// SIMATIC S7-200 project (STEP 7-Micro/WIN), CPU 224XP IE REL 02.01

SYMBOL_TABLE DI采集
急停               V0.0
单机/联机            V0.1
油泵启停             V0.2
1#进油启/停          V0.3
1#回油启/停          V0.4
2#进油启/停          V0.5
2#回油启/停          V0.6
缺相保护             V0.7
输入备用             V1.0
END_SYMBOL_TABLE

SYMBOL_TABLE DO控制
油泵_启             V22.0
1#进油_启           V20.2
1#回油_启           V20.4
1#卸荷_启           V20.6
2#进油_启           V21.0
2#回油_启           V21.2
2#卸荷_启           V21.4
备用_启             V21.6
油泵_停             V22.1
1#进油_停           V20.3
1#回油_停           V20.5
1#卸荷_停           V20.7
2#进油_停           V21.1
2#回油_停           V21.3
2#卸荷_停           V21.5
备用_停             V21.7
油泵_同             V41.0
1#进油_同           V40.1
1#回油_同           V40.2
1#卸荷_同           V40.3
2#进油_同           V40.4
2#回油_同           V40.5
2#卸荷_同           V40.6
备用_同             V40.7
END_SYMBOL_TABLE

SYMBOL_TABLE AI采集
AI1备用            VW50
AI2备用            VW52
1#压力             VW54
1#位移             VW56
2#压力             VW58
2#位移             VW60
压力1KN            VD78
压力2KN            VD86
压力量程上限           VW2000
位移量程上限           VW2002
AI1上限            VW2050
AI1下限            VW2052
AI2上限            VW2054
AI2下限            VW2056
1#压力L上限          VW2058
1#压力L下限          VW2060
1#位移L上限          VW2062
1#位移L下限          VW2064
2#压力L上限          VW2066
2#压力L下限          VW2068
2#位移L上限          VW2070
2#位移L下限          VW2072
AI1备用C           VW150
AI2备用C           VW152
1#压力C            VW154
1#位移C            VW156
2#压力C            VW158
2#位移C            VW160
1#压力断线           V100.0
1#位移断线           V100.1
2#压力断线           V100.2
2#位移断线           V100.3
END_SYMBOL_TABLE

SYMBOL_TABLE 故障
本机安全极限压力         VW2004
本机安全极限位移         VW2006
补压压力             VW2008
同步位移             VW2010
回程允许时间           VW2012
回程停机位移           VW2014
1#超本机压力_A        V2210.0
1#超本机位移_A        V2210.1
2#超本机压力_A        V2210.2
2#超本机位移_A        V2210.3
1#超安全压力_A        V2210.4
2#超安全压力_A        V2210.5
1#回程故障_A         V2210.6
2#回程故障_A         V2210.7
1#压力断线_A         V2211.0
1#位移断线_A         V2211.1
2#压力断线_A         V2211.2
2#位移断线_A         V2211.3
电机故障_A           V2211.4
总故障_A            V2211.7
END_SYMBOL_TABLE

SYMBOL_TABLE A1
A1设备标志           VW4018
A1第1B            VW4020
A1第2B            VW4022
A1第3B            VW4024
A1第4B            VW4026
A1第5B            VW4028
A1第6B            VW4030
A1终张B            VW4032
A1超张B            VW4034
A1回程B            VW4036
A1第1Y            VW4038
A1第2Y            VW4040
A1第3_1Y          VW4042
A1第3_2Y          VW4044
A1第4_1Y          VW4046
A1第4_2Y          VW4048
A1第5_1Y          VW4050
A1第5_2Y          VW4052
A1第6_1Y          VW4054
A1第6_2Y          VW4056
A1终张Y            VW4058
A1超张Y            VW4060
A1回程Y            VW4062
A1第1W            VW4064
A1第2W            VW4066
A1第3_1W          VW4068
A1第3_2W          VW4070
A1第4_1W          VW4072
A1第4_2W          VW4074
A1第5_1W          VW4076
A1第5_2W          VW4078
A1第6_1W          VW4080
A1第6_2W          VW4082
A1终张W            VW4084
A1超张W            VW4086
A1回程W            VW4088
A1安全B            VW4090
A1安全TJM          VW4092
A1设计油压M          VW4094
A1单根张拉力          VW4098
A1孔根数            VW4100
A1理论总伸长量         VW4102
A1理论总伸长上限        VW4104
A1理论总伸长下限        VW4106
A1实际伸长_mm        VW4112
A1单实际伸长_mm       VW4114
A1自控回程位移         VW4116
A1超张模式           VW4118
A1几次终张           VW4120
A1几顶拉            VW4122
A1顶选择            VW4124
A1是否终张           VW4126
A1理论回缩量（mm）      VW4128
A1张拉位置           VW4136
A1张拉控制力          VD4154
A1Y第1B           VW1300
A1Y第2B           VW1302
A1Y第3B           VW1304
A1Y第4B           VW1306
A1Y第5B           VW1308
A1Y第6B           VW1310
A1Y终张B           VW1312
A1Y超张B           VW1314
A1Y回程B           VW1316
A1Y安全B           VW1318
A1触发记录压力         VW2350
END_SYMBOL_TABLE

SYMBOL_TABLE 主控
卸荷完触发回程          M3.0
有卸荷标志            M1.0
回程停机缓冲位移         VW2016
伸长量不符合           V2212.3
参与机子到目标          V2220.0
A1_设置选择          V3124.0
B1_设置选择          V3124.1
A2_设置选择          V3124.2
B2_设置选择          V3124.3
持荷倒计时            VW2300
张拉位置最小值          VW2302
1组对拉位移最小值        VW2304
2组对拉位移最小值        VW2306
A1目标压力           VW2308
B1目标压力           VW2310
A2目标压力           VW2312
B2目标压力           VW2314
张拉中              V2206.0
回程中              V2206.1
持荷中              V2206.2
卸荷中              V2206.3
有无卸荷             VW2038
倒顶目标标志           V2212.0  // 1为第一次，0为第二进入
持荷完成标志           V2212.1
触发回程             V2212.2
A1伸长量不符合         V2212.4
B1伸长量不符合         V2212.5
A2伸长量不符合         V2212.6
B2伸长量不符合         V2212.7
位移超长触发回程         V2213.0
伸长量高于上限          V2213.1
A1伸长量高于上限        V2213.2
B1伸长量高于上限        V2213.3
A2伸长量高于上限        V2213.4
B2伸长量高于上限        V2213.5
算伸长量             V2213.6
伸长量已反算           V2213.7
自动进油_启           V2214.0
自动回油_启           V2214.1
自动卸荷_启           V2214.2
自动进油_停           V2215.0
自动回油_停           V2215.1
自动卸荷_停           V2215.2
自动进油_出           V2216.0
自动回油_出           V2216.1
自动卸荷_出           V2216.2
A1_实际选择          V2200.0
B1_实际选择          V2200.1
A2_实际选择          V2200.2
B2_实际选择          V2200.3
自动张拉             V2202.0
暂停张拉             V2202.1
手动进油             V2202.2
手动回油             V2202.3
A1到目标标志          V2218.0
B1到目标标志          V2218.1
A2到目标标志          V2218.2
B2到目标标志          V2218.3
A1自动进油_启         V2222.0
A1自动回油_启         V2222.1
A2自动进油_启         V2222.2
A2自动回油_启         V2222.3
A1自动进油_停         V2224.0
A1自动回油_停         V2224.1
A2自动进油_停         V2224.2
A2自动回油_停         V2224.3
A1自动卸荷_启         V2222.4
A2自动卸荷_启         V2222.5
A1自动卸荷_停         V2224.4
A2自动卸荷_停         V2224.5
A1自动进油_输出        V2226.0
A1自动回油_输出        V2226.1
A2自动进油_输出        V2226.2
A2自动回油_输出        V2226.3
A1自动卸荷_输出        V2226.4
A2自动卸荷_输出        V2226.5
A1回程到位           V2230.0
B1回程到位           V2230.1
A2回程到位           V2230.2
B2回程到位           V2230.3
A1卸荷到位           V2420.0
B1卸荷到位           V2420.1
A2卸荷到位           V2420.2
B2卸荷到位           V2420.3
总卸荷到位            V2420.4
A1触发记录           V2232.0
B1触发记录           V2232.1
A2触发记录           V2232.2
B2触发记录           V2232.3
触发写配方            V2232.4  // 触摸屏写完复位
调入已张拉的数据         V2204.0
新数据              V2204.1
调入模板数据           V2204.2
调入已张拉的数据_清       V2204.3
新数据_清            V2204.4
调入模板数据_清         V2204.5
调入已张拉的数据_触发      V2204.6
新数据_触发           V2204.7
调入模板数据_触发        V2205.0
总调入数据            V2205.7
A1回程触发           V2252.0
B1回程触发           V2252.1
A2回程触发           V2252.2
B2回程触发           V2252.3
复位超伸长量上限         V2250.0
复位超伸长量下限         V2250.1
持荷完成标志自锁2S       V2250.2
第一组实伸长量          VW2360
第二组实伸长量          VW2362
下载数据计时           VW2328
持荷时间             T37
张拉过标志            T38
回油时间             T39
故障复位时间           T40
写数据时间            T41
下载数据计时T          T42
持荷完成标志自锁2ST      T43
B1力值             VD2370
B2力值             VD2374
张回程完成标志          V2240.0
主启动油泵            V2254.0
主停止油泵            V2254.1
凋数据序号1           VW2390
凋数据序号2           VW2392
凋数据序号3           VW2394
凋数据序号4           VW2396
凋数据序号            VW2398
调入次数             VW2400
保存数据             V2208.0
不保存数据回程          V2208.1
未完成张拉保存数据回程      V2208.2
完成张拉超张保存数据回      V2208.3
触摸屏修改钢绞线根数       V2404.0
触摸屏修改张拉最大位移      V2404.1
触摸屏修改AB1伸长量      V2404.2
触摸屏修改AB2伸长量      V2404.3
单机频率             VW2120
张拉频率             VW2122
接近目标%            VW2124
目标频率%            VW2126
输出频率             VW2128
接近目标力            VD2130
副机张拉频率           VW2134
A1位移修正           VW2022
B1位移修正           VW2024
A2位移修正           VW2026
B2位移修正           VW2028
A1位移修正触发         VW2030
B1位移修正触发         VW2032
A2位移修正触发         VW2034
B2位移修正触发         VW2036
END_SYMBOL_TABLE

SYMBOL_TABLE 公共存储
G设备标志            VW3018
G第1B             VW3020
G第2B             VW3022
G第3B             VW3024
G第4B             VW3026
G第5B             VW3028
G第6B             VW3030
G终张B             VW3032
G超张B             VW3034
G回程B             VW3036
G第1Y             VW3038
G第2Y             VW3040
G第3_1Y           VW3042
G第3_2Y           VW3044
G第4_1Y           VW3046
G第4_2Y           VW3048
G第5_1Y           VW3050
G第5_2Y           VW3052
G第6_1Y           VW3054
G第6_2Y           VW3056
G终张Y             VW3058
G超张Y             VW3060
G回程Y             VW3062
G第1W             VW3064
G第2W             VW3066
G第3_1W           VW3068
G第3_2W           VW3070
G第4_1W           VW3072
G第4_2W           VW3074
G第5_1W           VW3076
G第5_2W           VW3078
G第6_1W           VW3080
G第6_2W           VW3082
G终张W             VW3084
G超张W             VW3086
G回程W             VW3088
G安全B             VW3090
G安全TJM           VW3092
G设计油压M           VW3094
G                VW3096
G单根张拉力           VW3098
G孔根数             VW3100
G理论总伸长量          VW3102
G理论总伸长上限         VW3104
G理论总伸长下限         VW3106
G实际伸长_mm         VW3112
G单实际伸长_mm        VW3114
G自控回程位移          VW3116
G超张模式            VW3118
G几次终张            VW3120
G几顶拉             VW3122   // 单拉 1对拉 2对拉
G顶选择             VW3124
G是否终张            VW3126
G理论回缩量（mm）       VW3128
G张拉控制力           VD3154
END_SYMBOL_TABLE

SYMBOL_TABLE B1
B1设备标志           VW4418
B1第1B            VW4420
B1第2B            VW4422
B1第3B            VW4424
B1第4B            VW4426
B1第5B            VW4428
B1第6B            VW4430
B1终张B            VW4432
B1超张B            VW4434
B1回程B            VW4436
B1第1Y            VW4438
B1第2Y            VW4440
B1第3_1Y          VW4442
B1第3_2Y          VW4444
B1第4_1Y          VW4446
B1第4_2Y          VW4448
B1第5_1Y          VW4450
B1第5_2Y          VW4452
B1第6_1Y          VW4454
B1第6_2Y          VW4456
B1终张Y            VW4458
B1超张Y            VW4460
B1回程Y            VW4462
B1第1W            VW4464
B1第2W            VW4466
B1第3_1W          VW4468
B1第3_2W          VW4470
B1第4_1W          VW4472
B1第4_2W          VW4474
B1第5_1W          VW4476
B1第5_2W          VW4478
B1第6_1W          VW4480
B1第6_2W          VW4482
B1终张W            VW4484
B1超张W            VW4486
B1回程W            VW4488
B1安全B            VW4490
B1安全TJM          VW4492
B1设计油压M          VW4494
B1单根张拉力          VW4498
B1孔根数            VW4500
B1理论总伸长量         VW4502
B1理论总伸长上限        VW4504
B1理论总伸长下限        VW4506
B1实际伸长_mm        VW4512
B1单实际伸长_mm       VW4514
B1自控回程位移         VW4516
B1超张模式           VW4518
B1几次终张           VW4520
B1几顶拉            VW4522
B1顶选择            VW4524
B1是否终张           VW4526
B1理论回缩量（mm）      VW4528
B1张拉控制力          VD4554
B1#压力            VW2610
B1#位移            VW2612
B2#压力            VW2614
B2#位移            VW2616
B1触发记录压力         VW2352
END_SYMBOL_TABLE

SYMBOL_TABLE A2
A2设备标志           VW4818
A2第1B            VW4820
A2第2B            VW4822
A2第3B            VW4824
A2第4B            VW4826
A2第5B            VW4828
A2第6B            VW4830
A2终张B            VW4832
A2超张B            VW4834
A2回程B            VW4836
A2第1Y            VW4838
A2第2Y            VW4840
A2第3_1Y          VW4842
A2第3_2Y          VW4844
A2第4_1Y          VW4846
A2第4_2Y          VW4848
A2第5_1Y          VW4850
A2第5_2Y          VW4852
A2第6_1Y          VW4854
A2第6_2Y          VW4856
A2终张Y            VW4858
A2超张Y            VW4860
A2回程Y            VW4862
A2第1W            VW4864
A2第2W            VW4866
A2第3_1W          VW4868
A2第3_2W          VW4870
A2第4_1W          VW4872
A2第4_2W          VW4874
A2第5_1W          VW4876
A2第5_2W          VW4878
A2第6_1W          VW4880
A2第6_2W          VW4882
A2终张W            VW4884
A2超张W            VW4886
A2回程W            VW4888
A2安全B            VW4890
A2安全TJM          VW4892
A2设计油压M          VW4894
A2单根张拉力          VW4898
A2孔根数            VW4900
A2理论总伸长量         VW4902
A2理论总伸长上限        VW4904
A2理论总伸长下限        VW4906
A2实际伸长_mm        VW4912
A2单实际伸长_mm       VW4914
A2自控回程位移         VW4916
A2超张模式           VW4918
A2几次终张           VW4920
A2几顶拉            VW4922
A2顶选择            VW4924
A2是否终张           VW4926
A2理论回缩量（mm）      VW4928
A2张拉位置           VW4936
A2张拉控制力          VD4954
A2触发记录压力         VW2354
END_SYMBOL_TABLE

SYMBOL_TABLE B2
B2设备标志           VW5218
B2第1B            VW5220
B2第2B            VW5222
B2第3B            VW5224
B2第4B            VW5226
B2第5B            VW5228
B2第6B            VW5230
B2终张B            VW5232
B2超张B            VW5234
B2回程B            VW5236
B2第1Y            VW5238
B2第2Y            VW5240
B2第3_1Y          VW5242
B2第3_2Y          VW5244
B2第4_1Y          VW5246
B2第4_2Y          VW5248
B2第5_1Y          VW5250
B2第5_2Y          VW5252
B2第6_1Y          VW5254
B2第6_2Y          VW5256
B2终张Y            VW5258
B2超张Y            VW5260
B2回程Y            VW5262
B2第1W            VW5264
B2第2W            VW5266
B2第3_1W          VW5268
B2第3_2W          VW5270
B2第4_1W          VW5272
B2第4_2W          VW5274
B2第5_1W          VW5276
B2第5_2W          VW5278
B2第6_1W          VW5280
B2第6_2W          VW5282
B2终张W            VW5284
B2超张W            VW5286
B2回程W            VW5288
B2安全B            VW5290
B2安全TJM          VW5292
B2设计油压M          VW5294
B2单根张拉力          VW5298
B2孔根数            VW5300
B2理论总伸长量         VW5302
B2理论总伸长上限        VW5304
B2理论总伸长下限        VW5306
B2实际伸长_mm        VW5312
B2单实际伸长_mm       VW5314
B2自控回程位移         VW5316
B2超张模式           VW5318
B2几次终张           VW5320
B2几顶拉            VW5322
B2顶选择            VW5324
B2是否终张           VW5326
B2理论回缩量（mm）      VW5328
B2张拉位置           VW5336
B2张拉控制力          VD5354
B2触发记录压力         VW2356
END_SYMBOL_TABLE

SYMBOL_TABLE mm
密码总错误            V8092.7
当前大于有效           V8092.2
当前小于记忆           V8092.1
有效年              VW8050
有效月              VW8052
有效日              VW8054
记忆年              VW8056
记忆月              VW8058
记忆日              VW8060
当前年              VW8062
当前月              VW8064
当前日              VW8066
校验错误             V8092.0
END_SYMBOL_TABLE

SYMBOL_TABLE 主副交换
副机通讯故障           V2402.1
B1到目标            V2604.0
B2到目标            V2604.1
FB1回程到位          V2604.2
FB2回程到位          V2604.3
B1卸荷到位F          V2604.4
B2卸荷到位F          V2604.5
B1目标%            VW2322
B2目标%            VW2326
触发回程位移           VW2018
B1安全压力           VW1418
B2安全压力           VW1618
F急停              V2600.0
单机_联机F           V2600.1
副油泵启动            V2600.2
副1进油启_停          V2600.3
F1回油启_停          V2600.4
F2进油启_停          V2600.5
F2回油启_停          V2600.6
F缺相保护            V2600.7
F油泵_Y            V2601.0
F1进油_Y           V2601.1
F1回油_Y           V2601.2
F1卸荷_Y           V2601.3
F2进油_Y           V2601.4
F2回油_Y           V2601.5
F2卸荷_Y           V2601.6
F备用_Y            V2601.7
END_SYMBOL_TABLE

SYMBOL_TABLE S7-200 符号
Always_On        SM0.0    // 始终接通为 ON
First_Scan_On    SM0.1    // 仅第一个扫描周期中接通为 ON
Clock_1s         SM0.5    // 在 1 秒钟的循环周期内，接通为 ON 0.5 秒，关断为 OFF 0.5  秒
Time_0_Intrvl    SMB34    // 定时中断 0 的时间间隔（从 1 至 255，以 1 毫秒为增量）。
END_SYMBOL_TABLE

ORGANIZATION_BLOCK 程序块:OB1
TITLE=程序注释
BEGIN
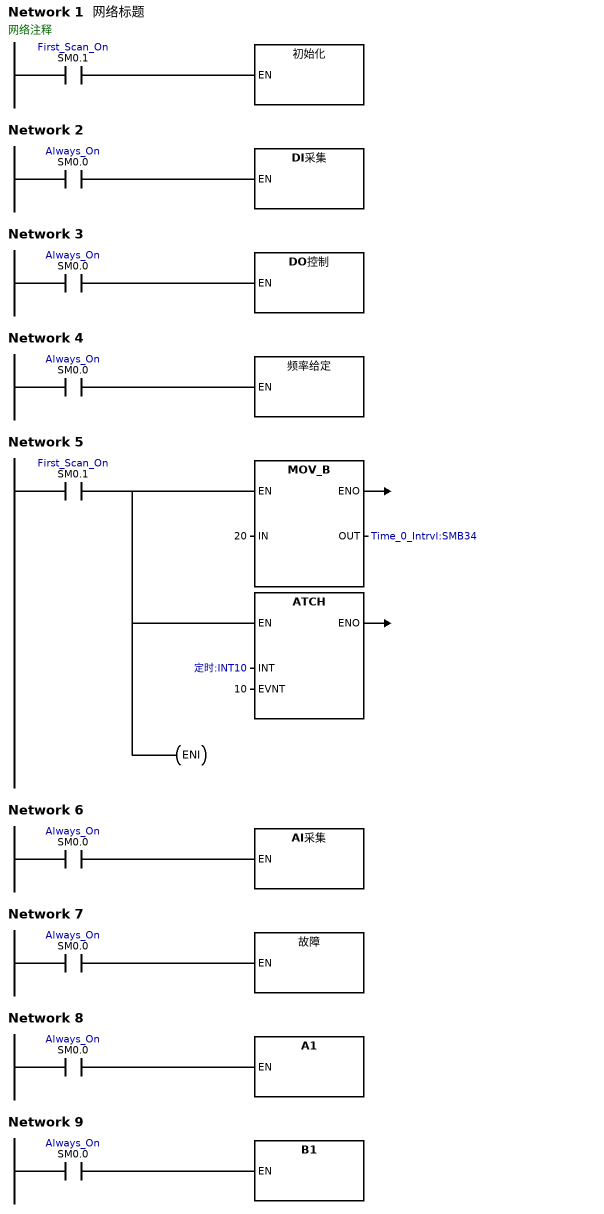
Network 1 // 网络标题
// 网络注释
LD     First_Scan_On:SM0.1
CALL   初始化:SBR0
Network 2
LD     Always_On:SM0.0
CALL   DI采集:SBR1
Network 3
LD     Always_On:SM0.0
CALL   DO控制:SBR2
Network 4
LD     Always_On:SM0.0
CALL   频率给定:SBR30
Network 5
LD     First_Scan_On:SM0.1
MOVB   20, Time_0_Intrvl:SMB34
ATCH   定时:INT10, 10
ENI
Network 6
LD     Always_On:SM0.0
CALL   AI采集:SBR3
Network 7
LD     Always_On:SM0.0
CALL   故障:SBR6
Network 8
LD     Always_On:SM0.0
CALL   A1:SBR7
Network 9
LD     Always_On:SM0.0
CALL   B1:SBR8
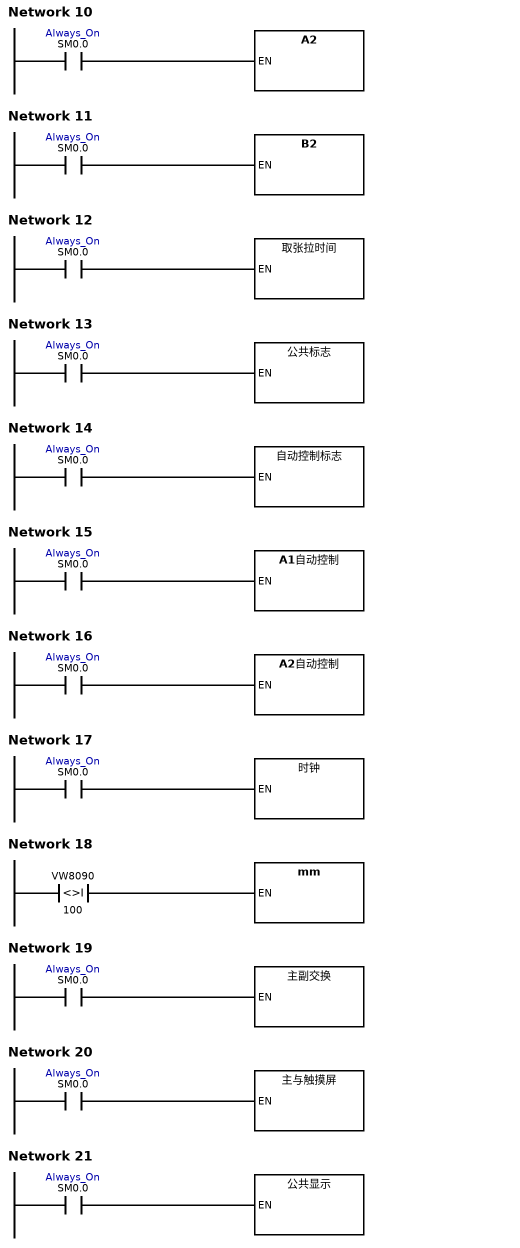
Network 10
LD     Always_On:SM0.0
CALL   A2:SBR9
Network 11
LD     Always_On:SM0.0
CALL   B2:SBR10
Network 12
LD     Always_On:SM0.0
CALL   取张拉时间:SBR28
Network 13
LD     Always_On:SM0.0
CALL   公共标志:SBR13
Network 14
LD     Always_On:SM0.0
CALL   自动控制标志:SBR14
Network 15
LD     Always_On:SM0.0
CALL   A1自动控制:SBR19
Network 16
LD     Always_On:SM0.0
CALL   A2自动控制:SBR20
Network 17
LD     Always_On:SM0.0
CALL   时钟:SBR21
Network 18
LDW<>  VW8090, 100
CALL   mm:SBR22
Network 19
LD     Always_On:SM0.0
CALL   主副交换:SBR23
Network 20
LD     Always_On:SM0.0
CALL   主与触摸屏:SBR18
Network 21
LD     Always_On:SM0.0
CALL   公共显示:SBR24
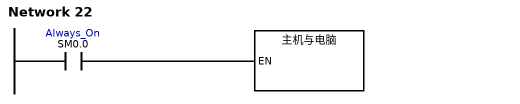
Network 22
LD     Always_On:SM0.0
CALL   主机与电脑:SBR29
END_ORGANIZATION_BLOCK

SUBROUTINE_BLOCK 初始化:SBR0
TITLE=
BEGIN
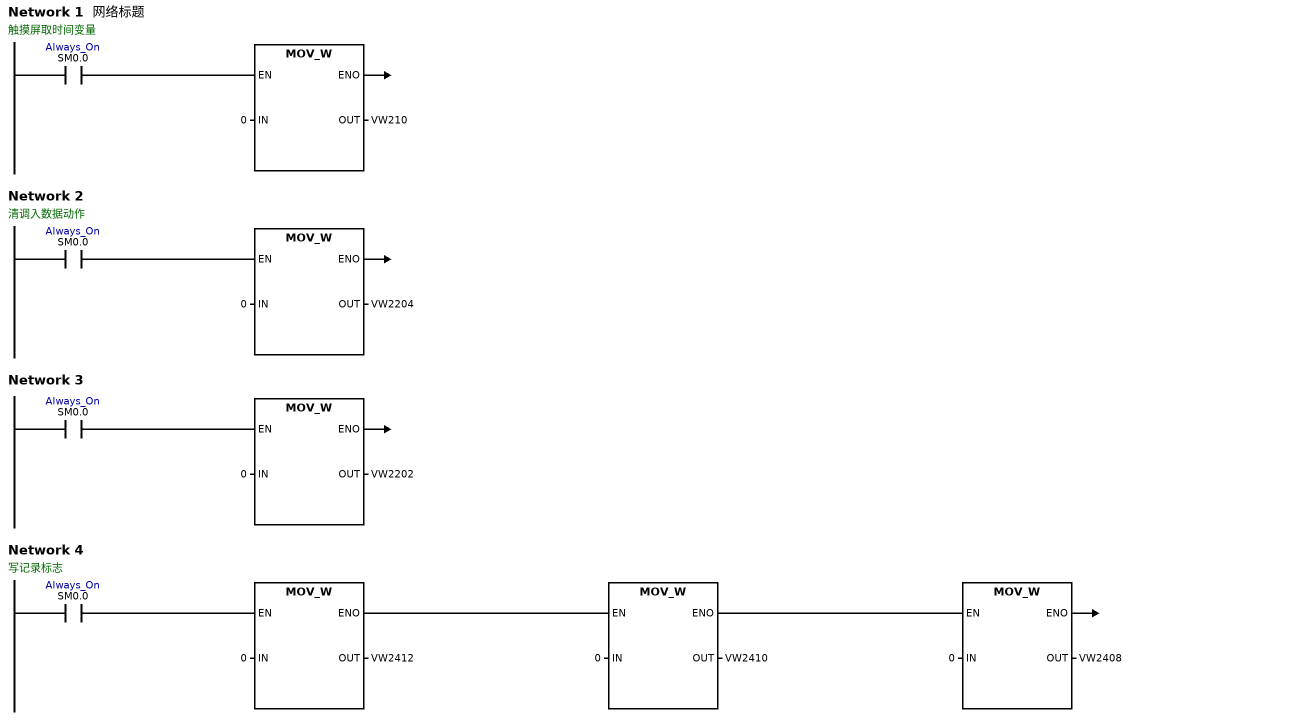
Network 1 // 网络标题
// 触摸屏取时间变量
LD     Always_On:SM0.0
MOVW   0, VW210
Network 2
// 清调入数据动作
LD     Always_On:SM0.0
MOVW   0, VW2204
Network 3
LD     Always_On:SM0.0
MOVW   0, VW2202
Network 4
// 写记录标志
LD     Always_On:SM0.0
MOVW   0, VW2412
AENO
MOVW   0, VW2410
AENO
MOVW   0, VW2408
END_SUBROUTINE_BLOCK

SUBROUTINE_BLOCK DI采集:SBR1
TITLE=
BEGIN
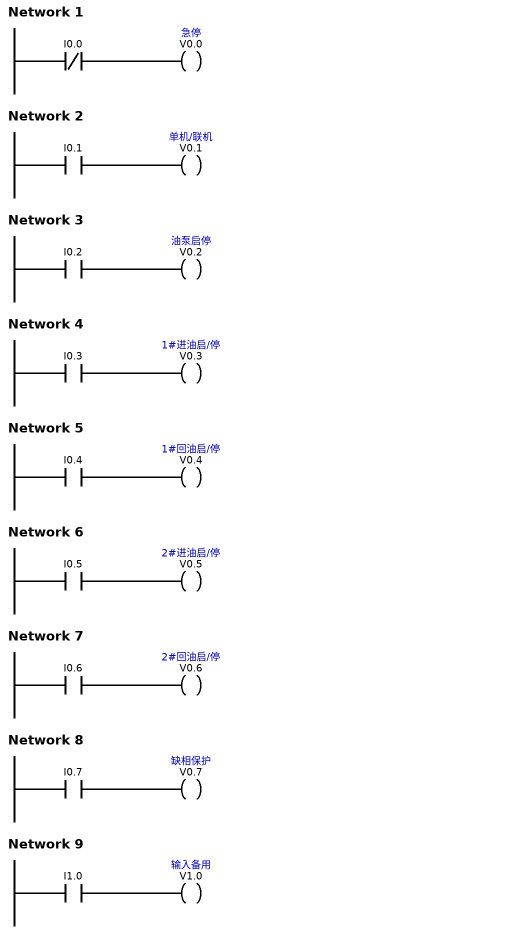
Network 1
LDN    I0.0
=      急停:V0.0
Network 2
LD     I0.1
=      单机/联机:V0.1
Network 3
LD     I0.2
=      油泵启停:V0.2
Network 4
LD     I0.3
=      1#进油启/停:V0.3
Network 5
LD     I0.4
=      1#回油启/停:V0.4
Network 6
LD     I0.5
=      2#进油启/停:V0.5
Network 7
LD     I0.6
=      2#回油启/停:V0.6
Network 8
LD     I0.7
=      缺相保护:V0.7
Network 9
LD     I1.0
=      输入备用:V1.0
END_SUBROUTINE_BLOCK

SUBROUTINE_BLOCK DO控制:SBR2
TITLE=
BEGIN
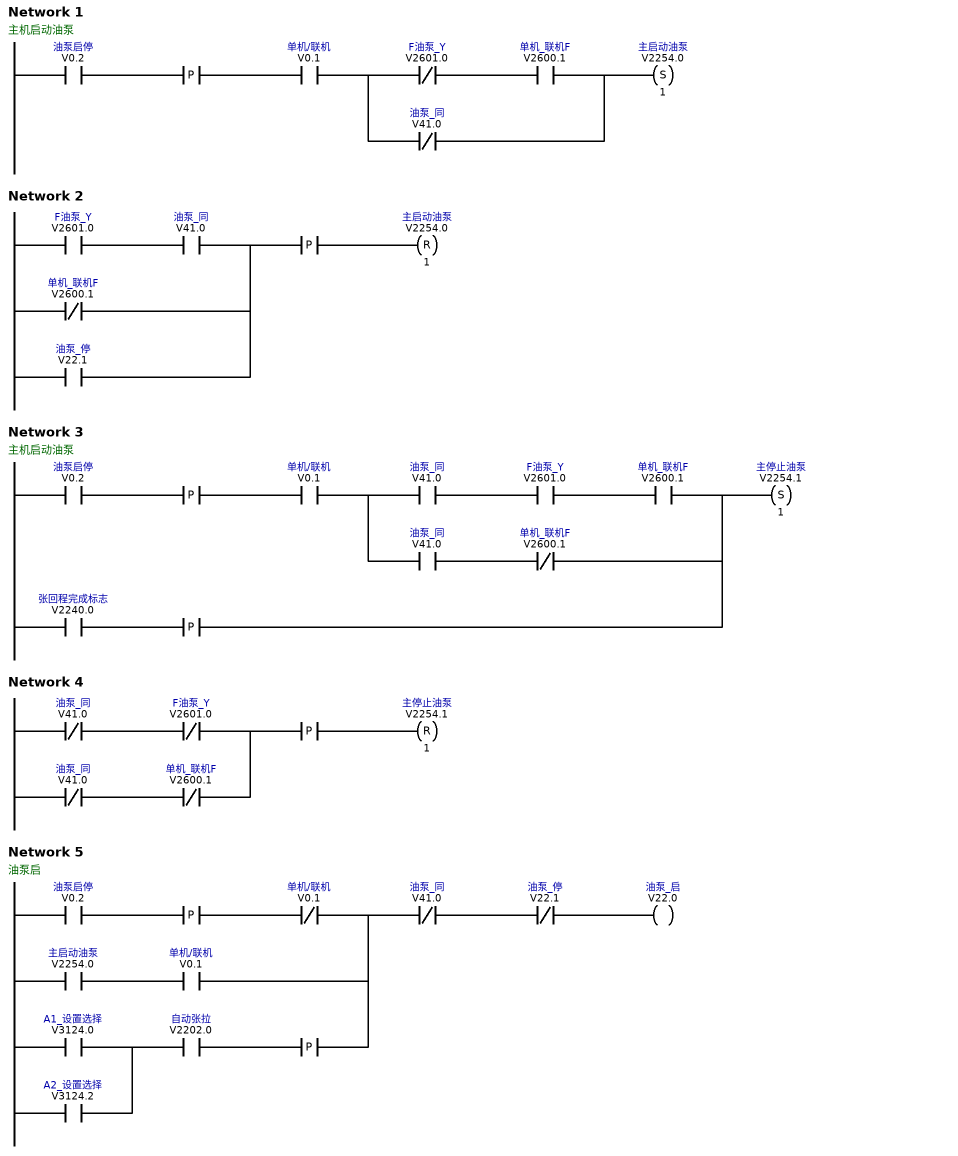
Network 1
// 主机启动油泵
LD     油泵启停:V0.2
EU
A      单机/联机:V0.1
LDN    F油泵_Y:V2601.0
A      单机_联机F:V2600.1
ON     油泵_同:V41.0
ALD
S      主启动油泵:V2254.0, 1
Network 2
LD     F油泵_Y:V2601.0
A      油泵_同:V41.0
ON     单机_联机F:V2600.1
O      油泵_停:V22.1
EU
R      主启动油泵:V2254.0, 1
Network 3
// 主机启动油泵
LD     油泵启停:V0.2
EU
A      单机/联机:V0.1
LD     油泵_同:V41.0
A      F油泵_Y:V2601.0
A      单机_联机F:V2600.1
LD     油泵_同:V41.0
AN     单机_联机F:V2600.1
OLD
ALD
LD     张回程完成标志:V2240.0
EU
OLD
S      主停止油泵:V2254.1, 1
Network 4
LDN    油泵_同:V41.0
AN     F油泵_Y:V2601.0
LDN    油泵_同:V41.0
AN     单机_联机F:V2600.1
OLD
EU
R      主停止油泵:V2254.1, 1
Network 5
// 油泵启
LD     油泵启停:V0.2
EU
AN     单机/联机:V0.1
LD     主启动油泵:V2254.0
A      单机/联机:V0.1
OLD
LD     A1_设置选择:V3124.0
O      A2_设置选择:V3124.2
A      自动张拉:V2202.0
EU
OLD
AN     油泵_同:V41.0
AN     油泵_停:V22.1
=      油泵_启:V22.0
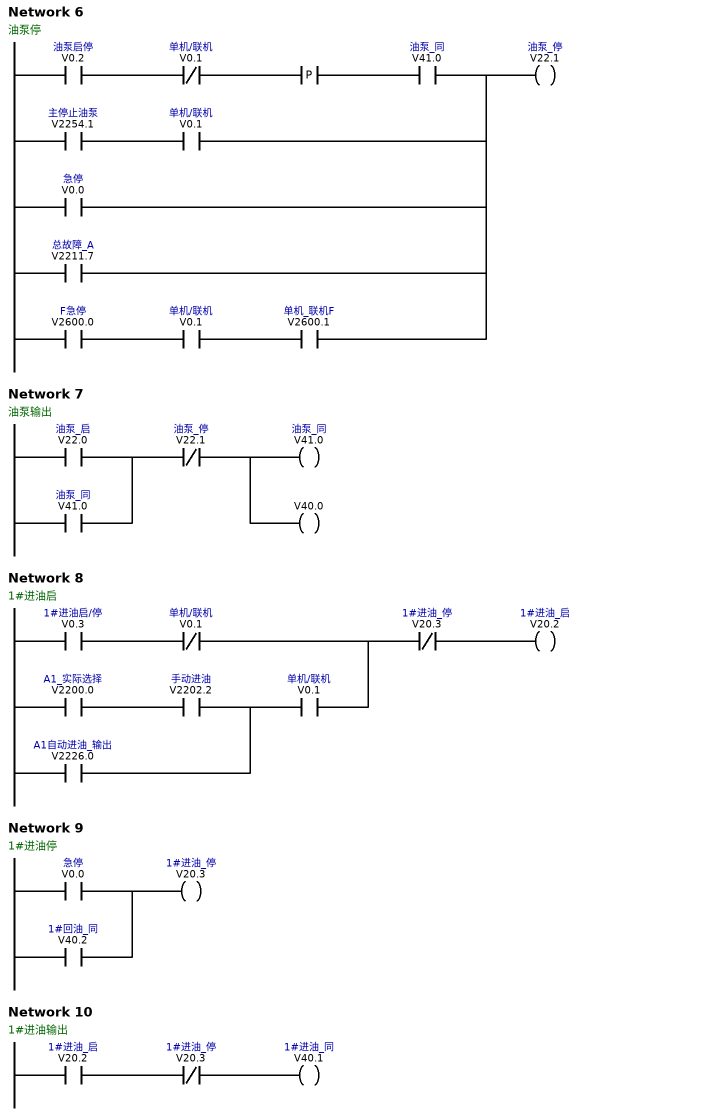
Network 6
// 油泵停
LD     油泵启停:V0.2
AN     单机/联机:V0.1
EU
A      油泵_同:V41.0
LD     主停止油泵:V2254.1
A      单机/联机:V0.1
OLD
O      急停:V0.0
O      总故障_A:V2211.7
LD     F急停:V2600.0
A      单机/联机:V0.1
A      单机_联机F:V2600.1
OLD
=      油泵_停:V22.1
Network 7
// 油泵输出
LD     油泵_启:V22.0
O      油泵_同:V41.0
AN     油泵_停:V22.1
=      油泵_同:V41.0
=      V40.0
Network 8
// 1#进油启
LD     1#进油启/停:V0.3
AN     单机/联机:V0.1
LD     A1_实际选择:V2200.0
A      手动进油:V2202.2
O      A1自动进油_输出:V2226.0
A      单机/联机:V0.1
OLD
AN     1#进油_停:V20.3
=      1#进油_启:V20.2
Network 9
// 1#进油停
LD     急停:V0.0
O      1#回油_同:V40.2
=      1#进油_停:V20.3
Network 10
// 1#进油输出
LD     1#进油_启:V20.2
AN     1#进油_停:V20.3
=      1#进油_同:V40.1
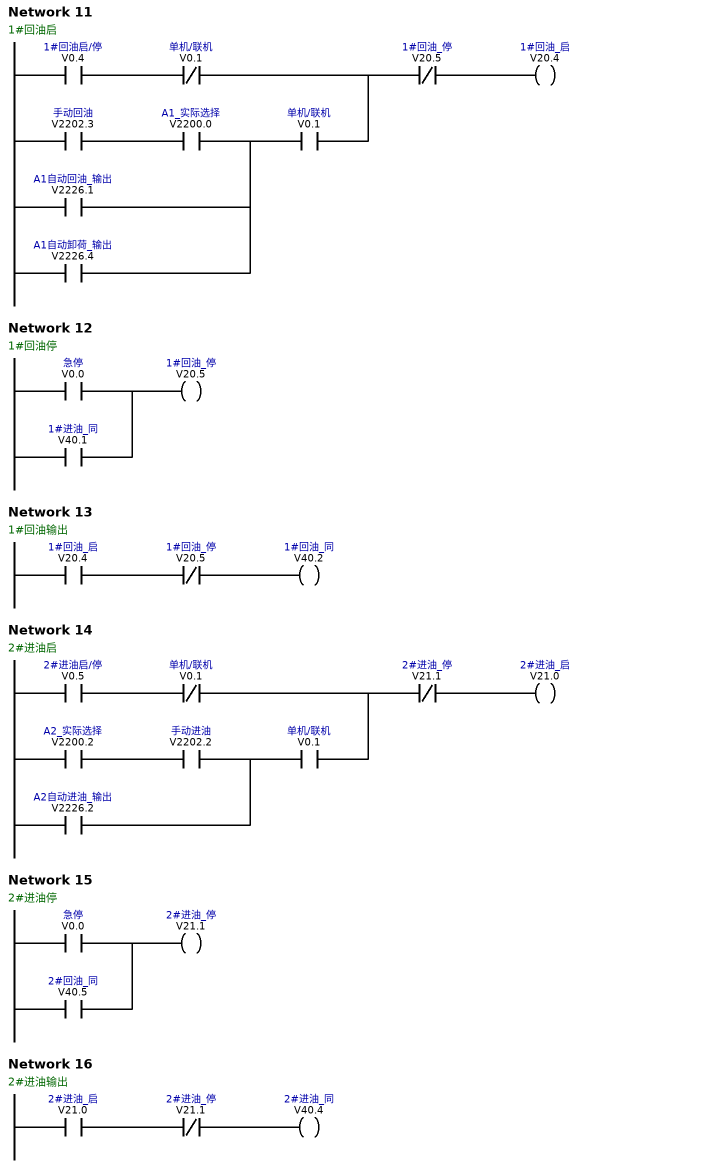
Network 11
// 1#回油启
LD     1#回油启/停:V0.4
AN     单机/联机:V0.1
LD     手动回油:V2202.3
A      A1_实际选择:V2200.0
O      A1自动回油_输出:V2226.1
O      A1自动卸荷_输出:V2226.4
A      单机/联机:V0.1
OLD
AN     1#回油_停:V20.5
=      1#回油_启:V20.4
Network 12
// 1#回油停
LD     急停:V0.0
O      1#进油_同:V40.1
=      1#回油_停:V20.5
Network 13
// 1#回油输出
LD     1#回油_启:V20.4
AN     1#回油_停:V20.5
=      1#回油_同:V40.2
Network 14
// 2#进油启
LD     2#进油启/停:V0.5
AN     单机/联机:V0.1
LD     A2_实际选择:V2200.2
A      手动进油:V2202.2
O      A2自动进油_输出:V2226.2
A      单机/联机:V0.1
OLD
AN     2#进油_停:V21.1
=      2#进油_启:V21.0
Network 15
// 2#进油停
LD     急停:V0.0
O      2#回油_同:V40.5
=      2#进油_停:V21.1
Network 16
// 2#进油输出
LD     2#进油_启:V21.0
AN     2#进油_停:V21.1
=      2#进油_同:V40.4
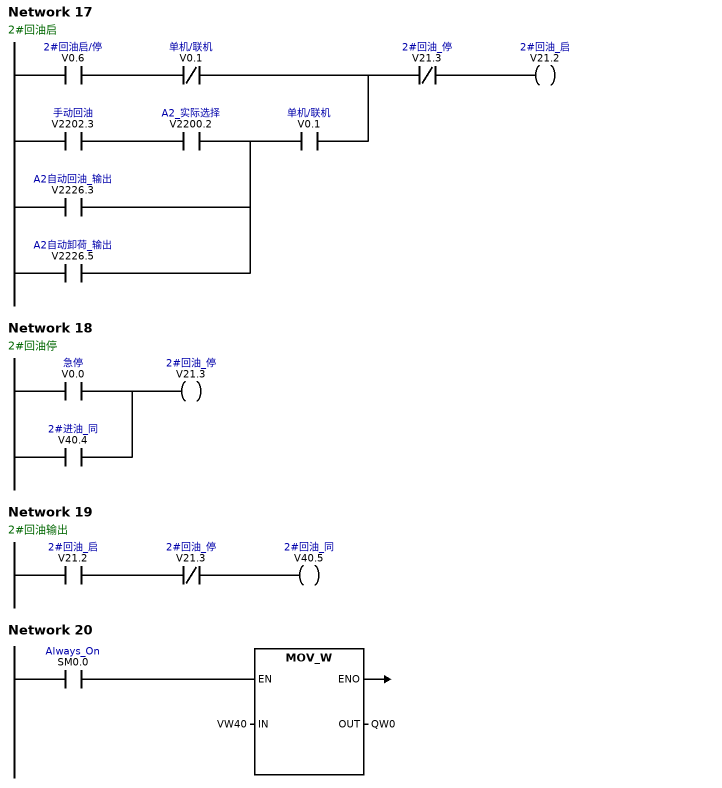
Network 17
// 2#回油启
LD     2#回油启/停:V0.6
AN     单机/联机:V0.1
LD     手动回油:V2202.3
A      A2_实际选择:V2200.2
O      A2自动回油_输出:V2226.3
O      A2自动卸荷_输出:V2226.5
A      单机/联机:V0.1
OLD
AN     2#回油_停:V21.3
=      2#回油_启:V21.2
Network 18
// 2#回油停
LD     急停:V0.0
O      2#进油_同:V40.4
=      2#回油_停:V21.3
Network 19
// 2#回油输出
LD     2#回油_启:V21.2
AN     2#回油_停:V21.3
=      2#回油_同:V40.5
Network 20
LD     Always_On:SM0.0
MOVW   VW40, QW0
END_SUBROUTINE_BLOCK

SUBROUTINE_BLOCK AI采集:SBR3
TITLE=
BEGIN
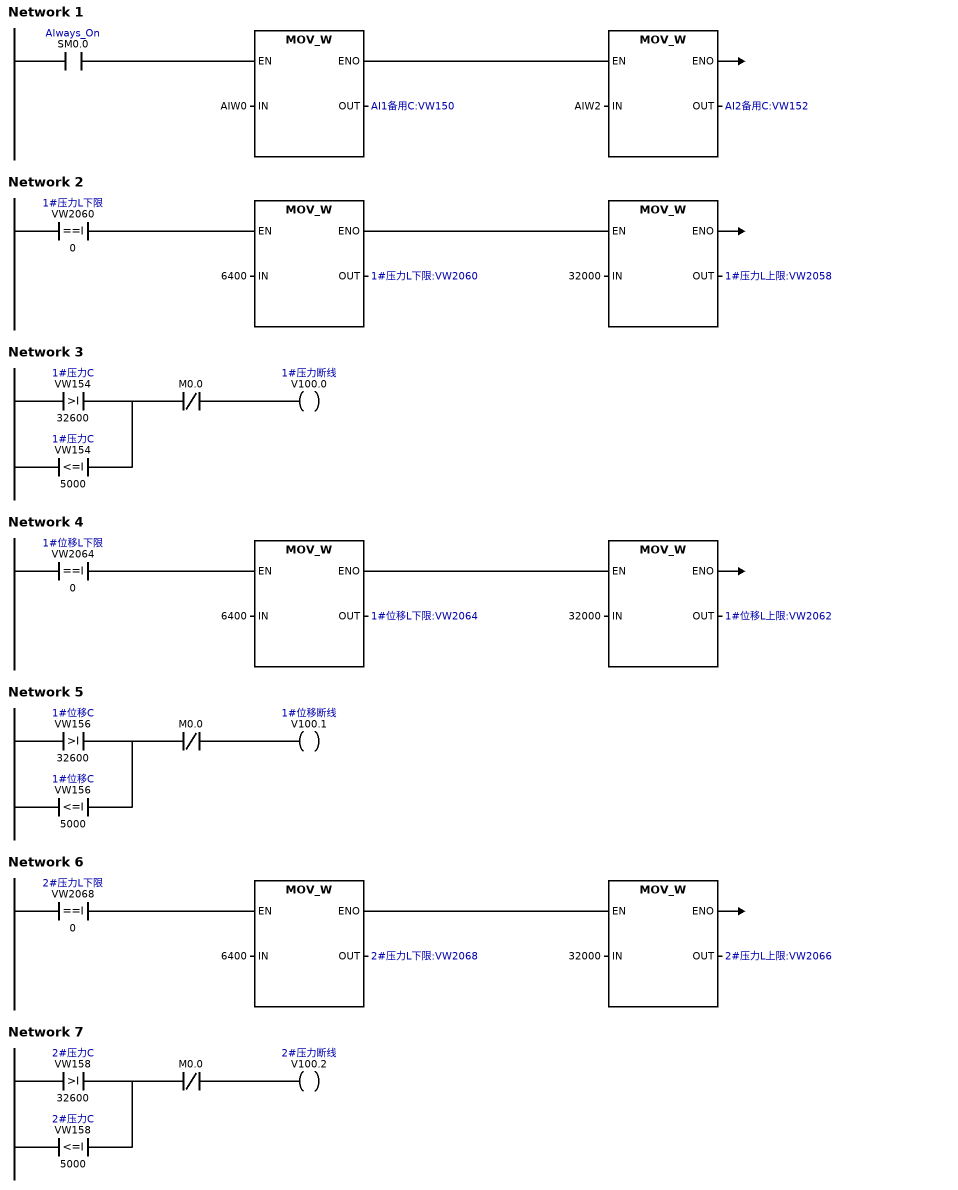
Network 1
LD     Always_On:SM0.0
MOVW   AIW0, AI1备用C:VW150
AENO
MOVW   AIW2, AI2备用C:VW152
Network 2
LDW=   1#压力L下限:VW2060, 0
MOVW   6400, 1#压力L下限:VW2060
AENO
MOVW   32000, 1#压力L上限:VW2058
Network 3
LDW>   1#压力C:VW154, 32600
OW<=   1#压力C:VW154, 5000
AN     M0.0
=      1#压力断线:V100.0
Network 4
LDW=   1#位移L下限:VW2064, 0
MOVW   6400, 1#位移L下限:VW2064
AENO
MOVW   32000, 1#位移L上限:VW2062
Network 5
LDW>   1#位移C:VW156, 32600
OW<=   1#位移C:VW156, 5000
AN     M0.0
=      1#位移断线:V100.1
Network 6
LDW=   2#压力L下限:VW2068, 0
MOVW   6400, 2#压力L下限:VW2068
AENO
MOVW   32000, 2#压力L上限:VW2066
Network 7
LDW>   2#压力C:VW158, 32600
OW<=   2#压力C:VW158, 5000
AN     M0.0
=      2#压力断线:V100.2
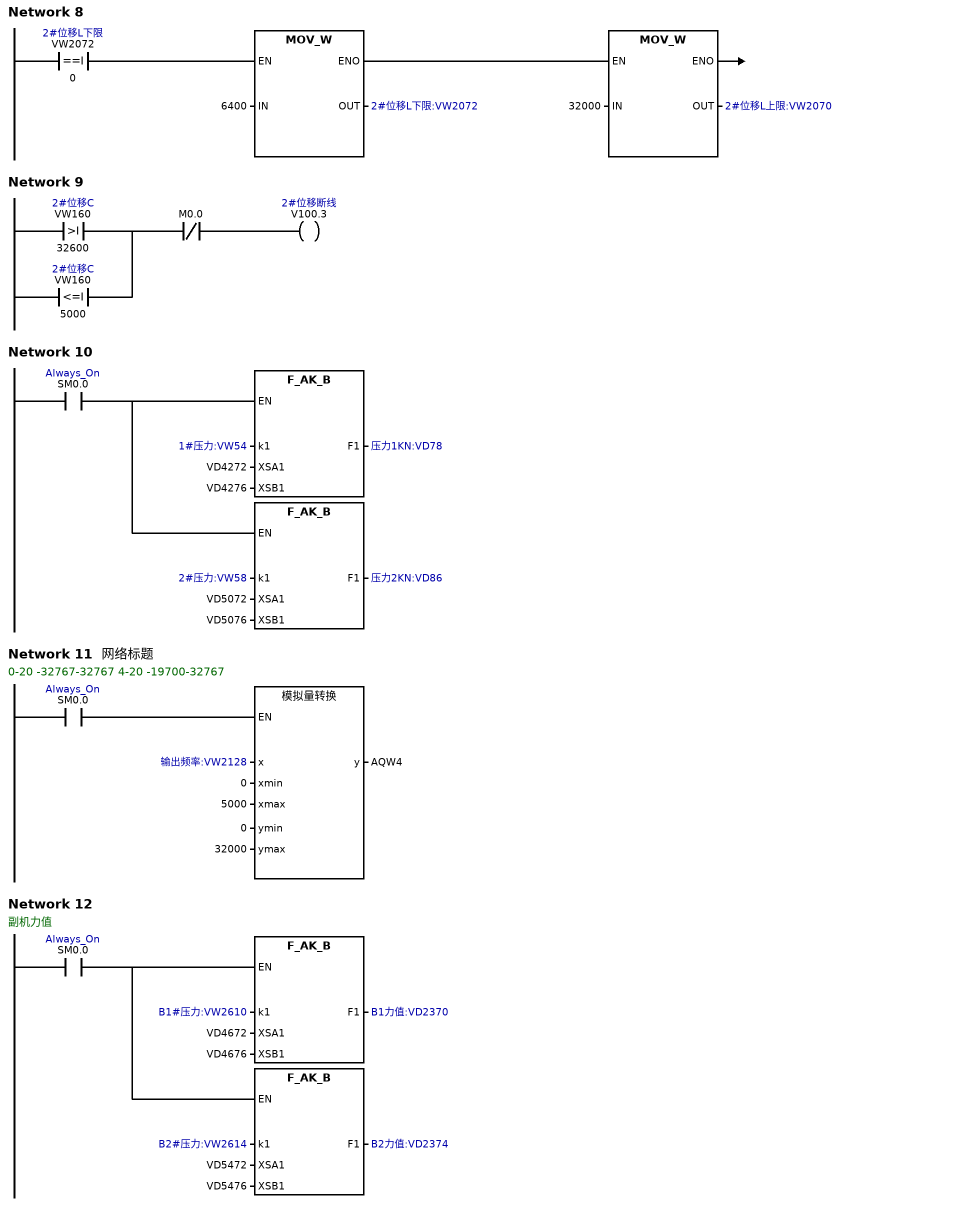
Network 8
LDW=   2#位移L下限:VW2072, 0
MOVW   6400, 2#位移L下限:VW2072
AENO
MOVW   32000, 2#位移L上限:VW2070
Network 9
LDW>   2#位移C:VW160, 32600
OW<=   2#位移C:VW160, 5000
AN     M0.0
=      2#位移断线:V100.3
Network 10
LD     Always_On:SM0.0
CALL   F_AK_B:SBR26, 1#压力:VW54, VD4272, VD4276, 压力1KN:VD78
CALL   F_AK_B:SBR26, 2#压力:VW58, VD5072, VD5076, 压力2KN:VD86
Network 11 // 网络标题
// 0-20 -32767-32767 4-20 -19700-32767
LD     Always_On:SM0.0
CALL   模拟量转换:SBR4, 输出频率:VW2128, 0, 5000, 0, 32000, AQW4
Network 12
// 副机力值
LD     Always_On:SM0.0
CALL   F_AK_B:SBR26, B1#压力:VW2610, VD4672, VD4676, B1力值:VD2370
CALL   F_AK_B:SBR26, B2#压力:VW2614, VD5472, VD5476, B2力值:VD2374
END_SUBROUTINE_BLOCK

SUBROUTINE_BLOCK 模拟量转换:SBR4
TITLE=
VAR_INPUT
x:INT;	// LW0 输入值
xmin:INT;	// LW2 输入最小值
xmax:INT;	// LW4 输入最大值
ymin:INT;	// LW6 输出最小值
ymax:INT;	// LW8 输出最大值
END_VAR
VAR_OUTPUT
y:INT;	// LW10 输出值
END_VAR
VAR
X3:REAL;	// LD12 
XMIN3:REAL;	// LD16 
XMAX3:REAL;	// LD20 
YMIN3:REAL;	// LD24 
YMAX3:REAL;	// LD28 
a1:REAL;	// LD32 
b1:REAL;	// LD36 
y2:DINT;	// LD40 
SZZJ1:DINT;	// LD44 双整中间变量
SZZJ2:DINT;	// LD48 
SZZJ3:DINT;	// LD52 
SZZJ4:DINT;	// LD56 
END_VAR
BEGIN
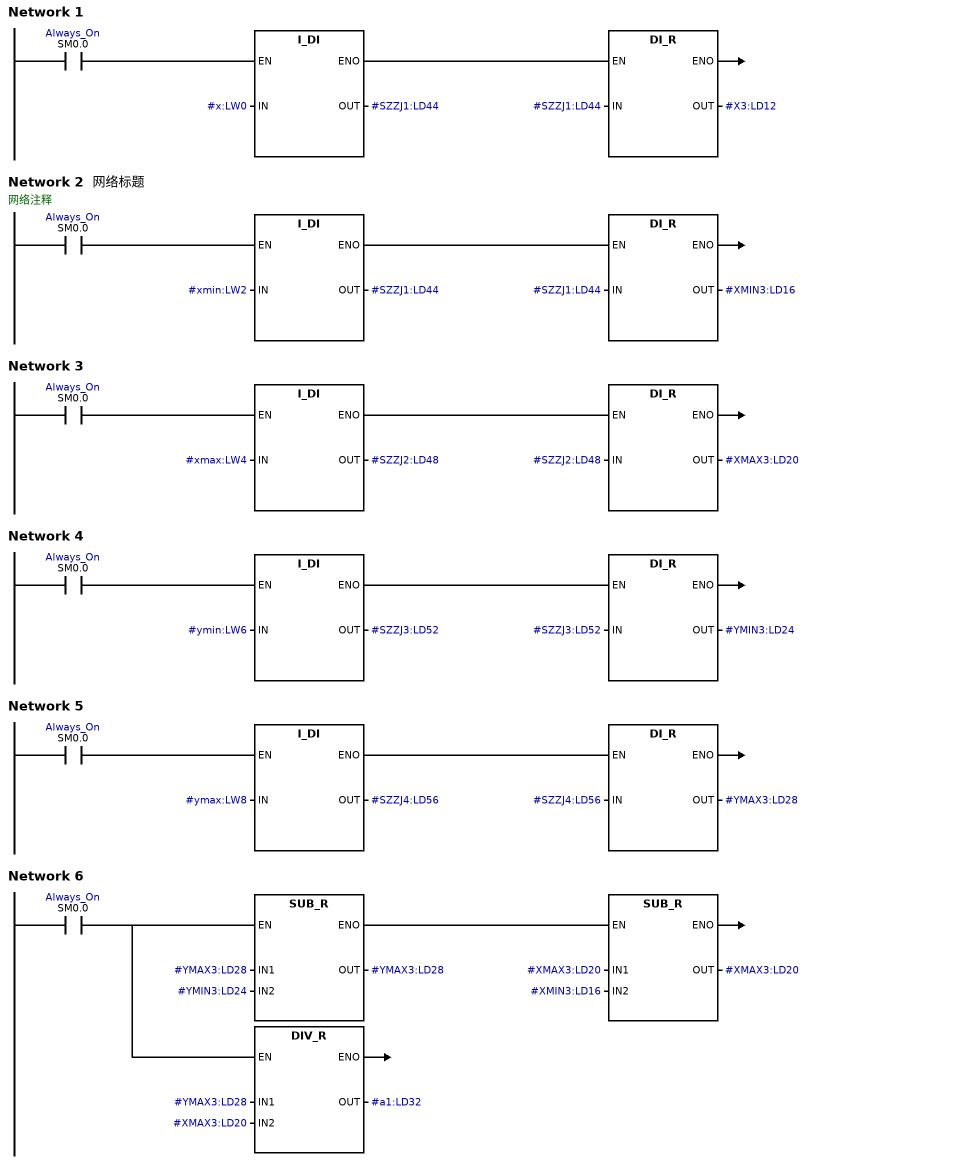
Network 1
LD     Always_On:SM0.0
ITD    #x:LW0, #SZZJ1:LD44
AENO
DTR    #SZZJ1:LD44, #X3:LD12
Network 2 // 网络标题
// 网络注释
LD     Always_On:SM0.0
ITD    #xmin:LW2, #SZZJ1:LD44
AENO
DTR    #SZZJ1:LD44, #XMIN3:LD16
Network 3
LD     Always_On:SM0.0
ITD    #xmax:LW4, #SZZJ2:LD48
AENO
DTR    #SZZJ2:LD48, #XMAX3:LD20
Network 4
LD     Always_On:SM0.0
ITD    #ymin:LW6, #SZZJ3:LD52
AENO
DTR    #SZZJ3:LD52, #YMIN3:LD24
Network 5
LD     Always_On:SM0.0
ITD    #ymax:LW8, #SZZJ4:LD56
AENO
DTR    #SZZJ4:LD56, #YMAX3:LD28
Network 6
LD     Always_On:SM0.0
LPS
-R     #YMIN3:LD24, #YMAX3:LD28
AENO
-R     #XMIN3:LD16, #XMAX3:LD20
LPP
MOVR   #YMAX3:LD28, #a1:LD32
/R     #XMAX3:LD20, #a1:LD32
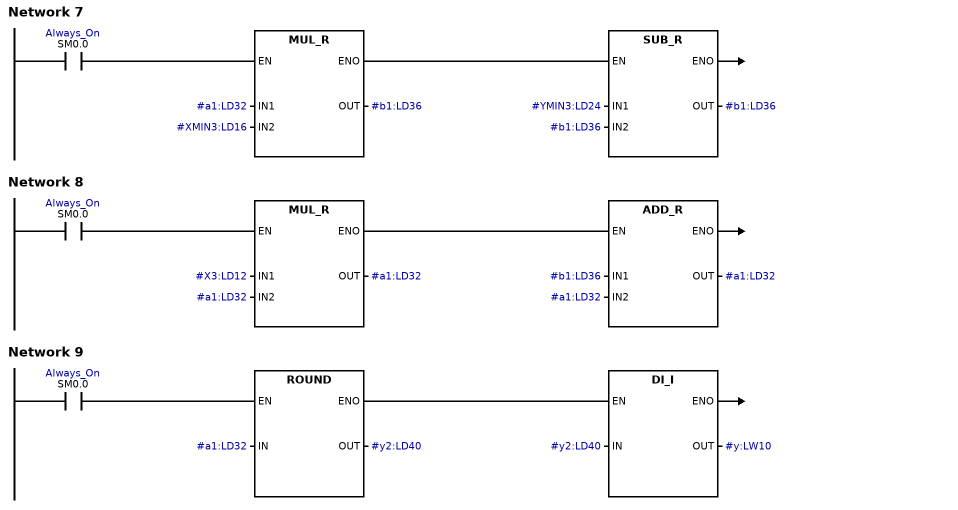
Network 7
LD     Always_On:SM0.0
MOVR   #a1:LD32, #b1:LD36
AENO
*R     #XMIN3:LD16, #b1:LD36
AENO
*R     -1.0, #b1:LD36
+R     #YMIN3:LD24, #b1:LD36
Network 8
LD     Always_On:SM0.0
*R     #X3:LD12, #a1:LD32
AENO
+R     #b1:LD36, #a1:LD32
Network 9
LD     Always_On:SM0.0
ROUND  #a1:LD32, #y2:LD40
AENO
DTI    #y2:LD40, #y:LW10
END_SUBROUTINE_BLOCK

SUBROUTINE_BLOCK 整数转实数:SBR5
TITLE=
VAR_INPUT
A1:INT;	// LW0 
END_VAR
VAR_OUTPUT
A3:REAL;	// LD2 
END_VAR
VAR
A2:DINT;	// LD6 
END_VAR
BEGIN
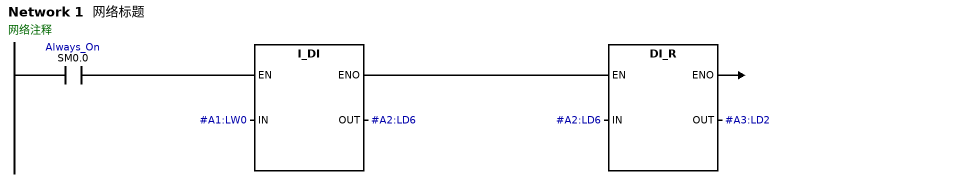
Network 1 // 网络标题
// 网络注释
LD     Always_On:SM0.0
ITD    #A1:LW0, #A2:LD6
AENO
DTR    #A2:LD6, #A3:LD2
END_SUBROUTINE_BLOCK

SUBROUTINE_BLOCK 故障:SBR6
TITLE=子程序注释
BEGIN
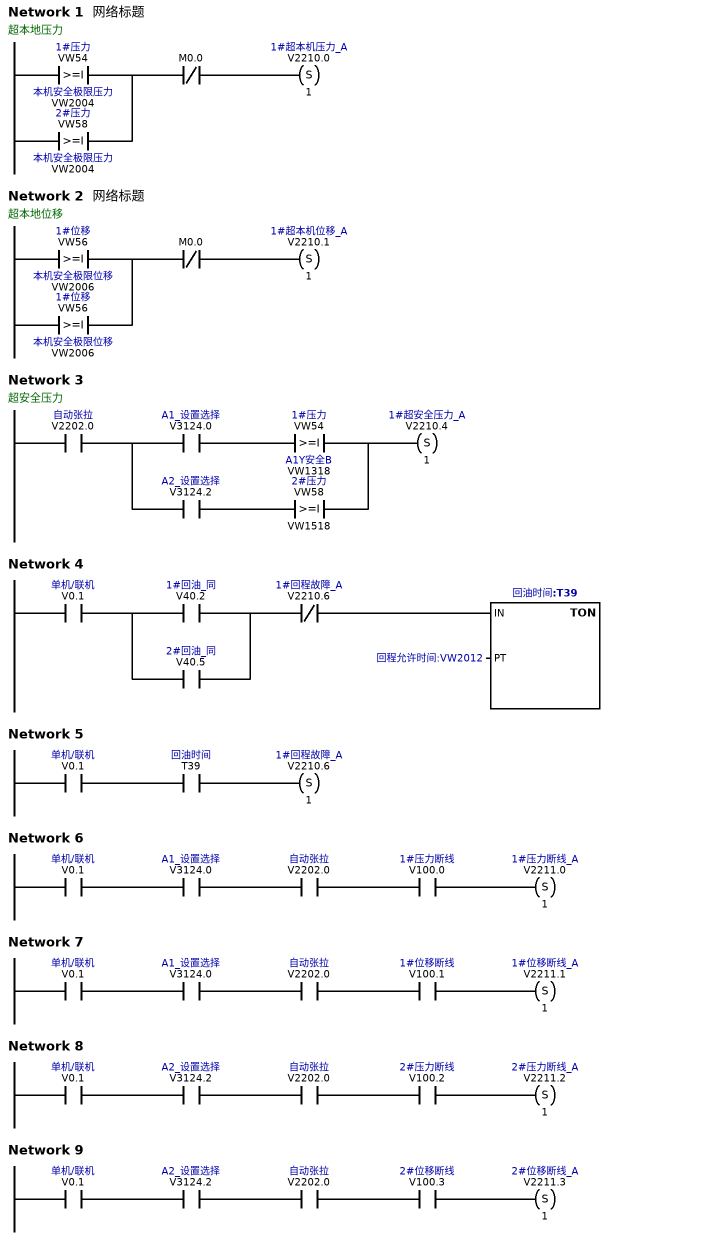
Network 1 // 网络标题
// 超本地压力
LDW>=  1#压力:VW54, 本机安全极限压力:VW2004
OW>=   2#压力:VW58, 本机安全极限压力:VW2004
AN     M0.0
S      1#超本机压力_A:V2210.0, 1
Network 2 // 网络标题
// 超本地位移
LDW>=  1#位移:VW56, 本机安全极限位移:VW2006
OW>=   1#位移:VW56, 本机安全极限位移:VW2006
AN     M0.0
S      1#超本机位移_A:V2210.1, 1
Network 3
// 超安全压力
LD     自动张拉:V2202.0
LD     A1_设置选择:V3124.0
AW>=   1#压力:VW54, A1Y安全B:VW1318
LD     A2_设置选择:V3124.2
AW>=   2#压力:VW58, VW1518
OLD
ALD
S      1#超安全压力_A:V2210.4, 1
Network 4
LD     单机/联机:V0.1
LD     1#回油_同:V40.2
O      2#回油_同:V40.5
ALD
AN     1#回程故障_A:V2210.6
TON    回油时间:T39, 回程允许时间:VW2012
Network 5
LD     单机/联机:V0.1
A      回油时间:T39
S      1#回程故障_A:V2210.6, 1
Network 6
LD     单机/联机:V0.1
A      A1_设置选择:V3124.0
A      自动张拉:V2202.0
A      1#压力断线:V100.0
S      1#压力断线_A:V2211.0, 1
Network 7
LD     单机/联机:V0.1
A      A1_设置选择:V3124.0
A      自动张拉:V2202.0
A      1#位移断线:V100.1
S      1#位移断线_A:V2211.1, 1
Network 8
LD     单机/联机:V0.1
A      A2_设置选择:V3124.2
A      自动张拉:V2202.0
A      2#压力断线:V100.2
S      2#压力断线_A:V2211.2, 1
Network 9
LD     单机/联机:V0.1
A      A2_设置选择:V3124.2
A      自动张拉:V2202.0
A      2#位移断线:V100.3
S      2#位移断线_A:V2211.3, 1
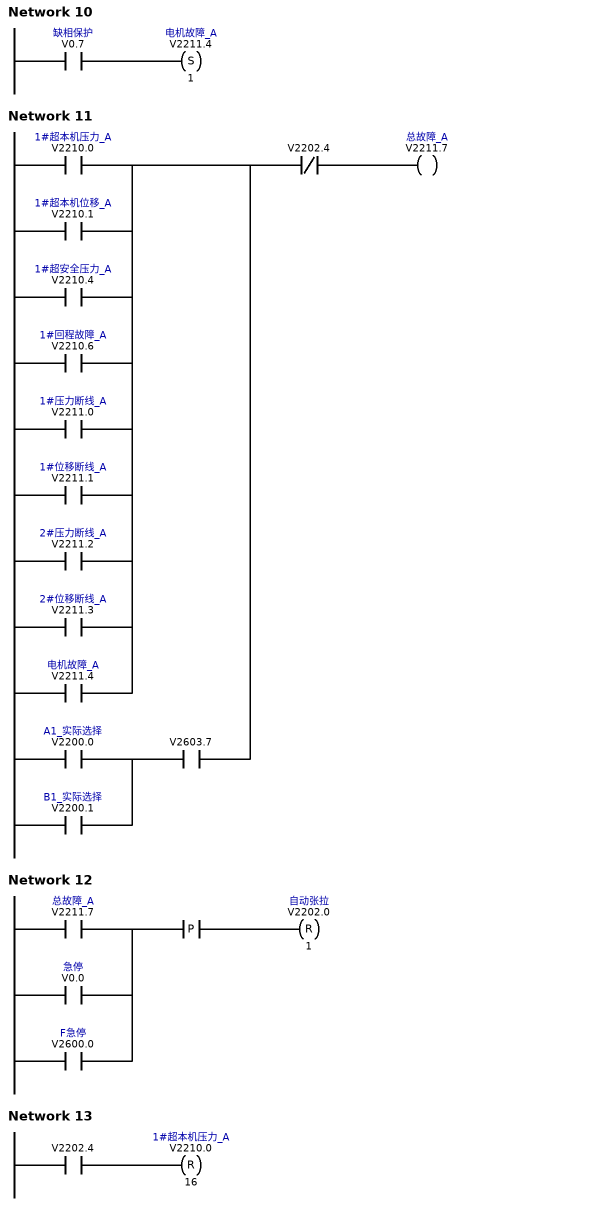
Network 10
LD     缺相保护:V0.7
S      电机故障_A:V2211.4, 1
Network 11
LD     1#超本机压力_A:V2210.0
O      1#超本机位移_A:V2210.1
O      1#超安全压力_A:V2210.4
O      1#回程故障_A:V2210.6
O      1#压力断线_A:V2211.0
O      1#位移断线_A:V2211.1
O      2#压力断线_A:V2211.2
O      2#位移断线_A:V2211.3
O      电机故障_A:V2211.4
LD     A1_实际选择:V2200.0
O      B1_实际选择:V2200.1
A      V2603.7
OLD
AN     V2202.4
=      总故障_A:V2211.7
Network 12
LD     总故障_A:V2211.7
O      急停:V0.0
O      F急停:V2600.0
EU
R      自动张拉:V2202.0, 1
Network 13
LD     V2202.4
R      1#超本机压力_A:V2210.0, 16
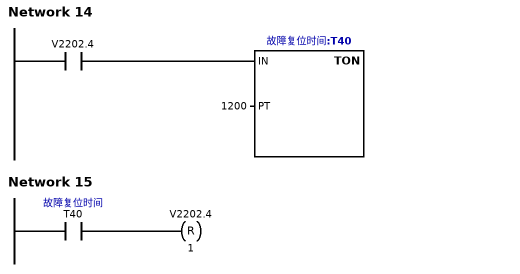
Network 14
LD     V2202.4
TON    故障复位时间:T40, 1200
Network 15
LD     故障复位时间:T40
R      V2202.4, 1
END_SUBROUTINE_BLOCK

// SBR7: protected block, not included

// SBR8: protected block, not included

// SBR9: protected block, not included

// SBR10: protected block, not included

SUBROUTINE_BLOCK 算目标压力:SBR11
TITLE=子程序注释
VAR_INPUT
百分比:INT;	// LW0 
控制力:REAL;	// LD2 
系数a1:REAL;	// LD6 
系数b1:REAL;	// LD10 
END_VAR
VAR_OUTPUT
输出压力:INT;	// LW14 
END_VAR
VAR
百分比控制力:REAL;	// LD16 
实转双整:DINT;	// LD20 
END_VAR
BEGIN
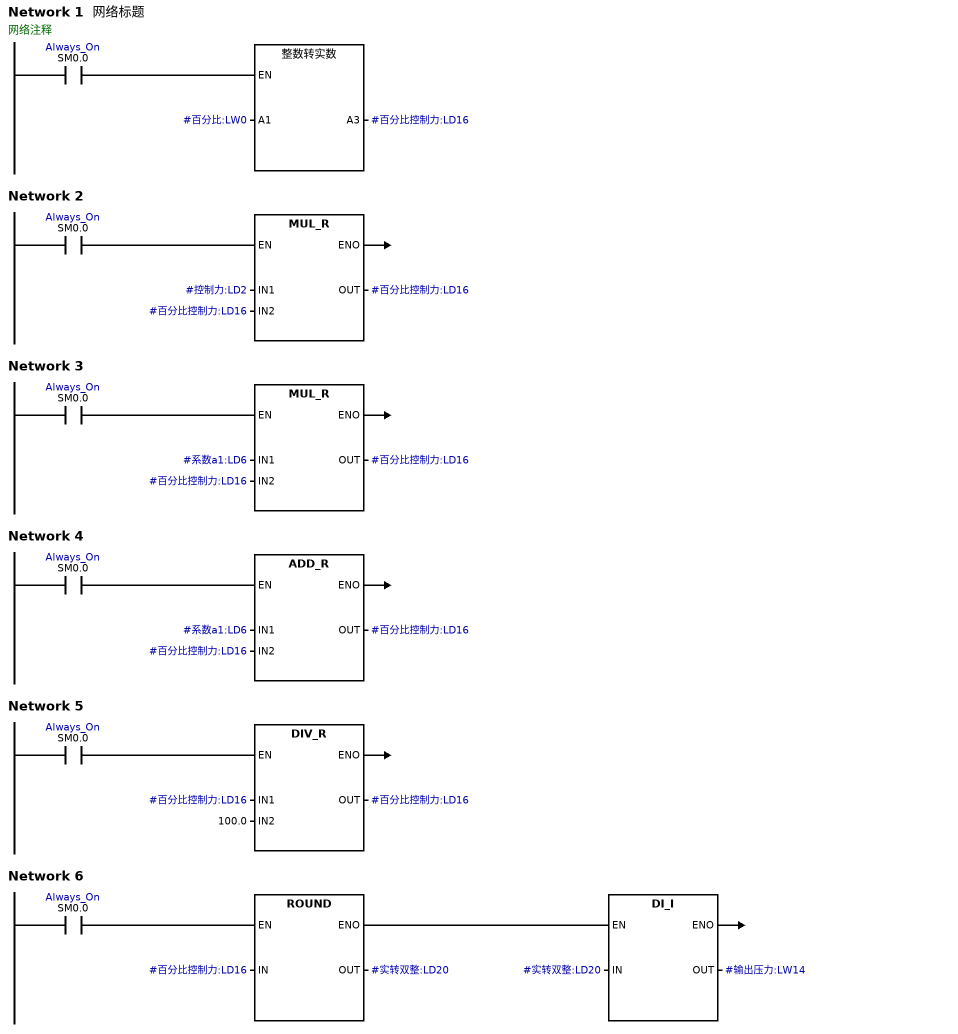
Network 1 // 网络标题
// 网络注释
LD     Always_On:SM0.0
CALL   整数转实数:SBR5, #百分比:LW0, #百分比控制力:LD16
Network 2
LD     Always_On:SM0.0
*R     #控制力:LD2, #百分比控制力:LD16
Network 3
LD     Always_On:SM0.0
*R     #系数a1:LD6, #百分比控制力:LD16
Network 4
LD     Always_On:SM0.0
+R     #系数a1:LD6, #百分比控制力:LD16
Network 5
LD     Always_On:SM0.0
/R     100.0, #百分比控制力:LD16
Network 6
LD     Always_On:SM0.0
ROUND  #百分比控制力:LD16, #实转双整:LD20
AENO
DTI    #实转双整:LD20, #输出压力:LW14
END_SUBROUTINE_BLOCK

SUBROUTINE_BLOCK 取最小值:SBR12
TITLE=子程序注释
VAR_INPUT
A1_IN:WORD;	// LW0 
B1_IN:WORD;	// LW2 
A2_IN:WORD;	// LW4 
B2_IN:WORD;	// LW6 
END_VAR
VAR_OUTPUT
最小值:WORD;	// LW8 
END_VAR
VAR
A1张拉目标:WORD;	// LW10 
B1张拉目标:WORD;	// LW12 
A2张拉目标:WORD;	// LW14 
B2张拉目标:WORD;	// LW16 
比较最小值:WORD;	// LW18 
END_VAR
BEGIN
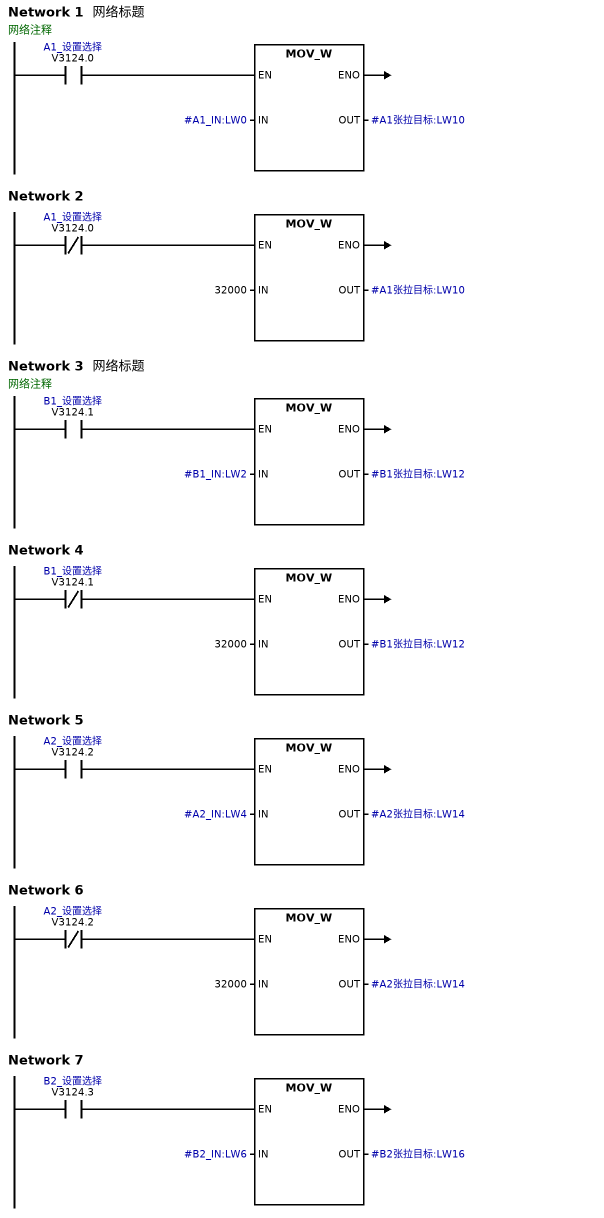
Network 1 // 网络标题
// 网络注释
LD     A1_设置选择:V3124.0
MOVW   #A1_IN:LW0, #A1张拉目标:LW10
Network 2
LDN    A1_设置选择:V3124.0
MOVW   32000, #A1张拉目标:LW10
Network 3 // 网络标题
// 网络注释
LD     B1_设置选择:V3124.1
MOVW   #B1_IN:LW2, #B1张拉目标:LW12
Network 4
LDN    B1_设置选择:V3124.1
MOVW   32000, #B1张拉目标:LW12
Network 5
LD     A2_设置选择:V3124.2
MOVW   #A2_IN:LW4, #A2张拉目标:LW14
Network 6
LDN    A2_设置选择:V3124.2
MOVW   32000, #A2张拉目标:LW14
Network 7
LD     B2_设置选择:V3124.3
MOVW   #B2_IN:LW6, #B2张拉目标:LW16
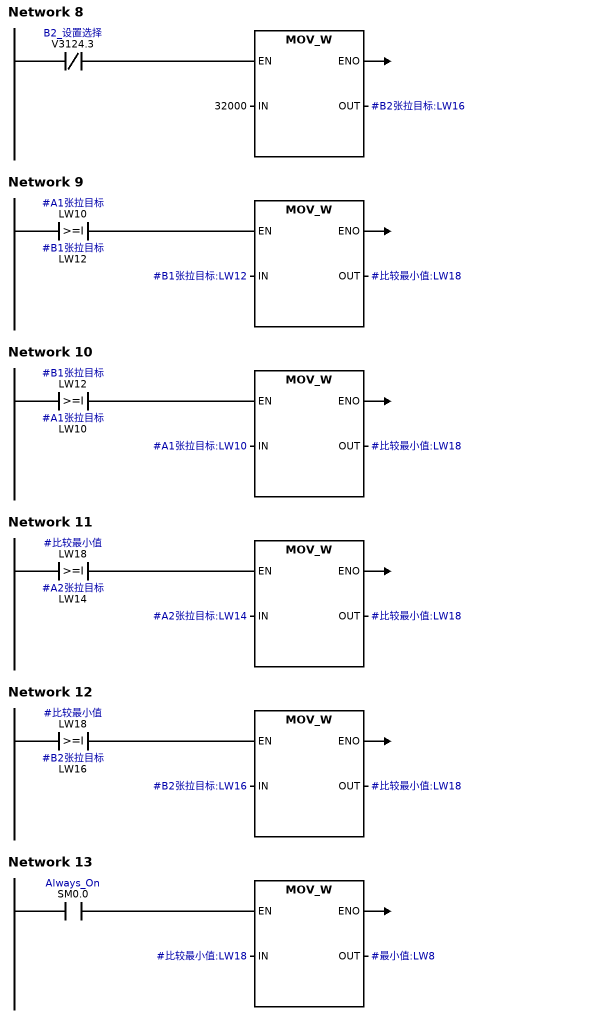
Network 8
LDN    B2_设置选择:V3124.3
MOVW   32000, #B2张拉目标:LW16
Network 9
LDW>=  #A1张拉目标:LW10, #B1张拉目标:LW12
MOVW   #B1张拉目标:LW12, #比较最小值:LW18
Network 10
LDW>=  #B1张拉目标:LW12, #A1张拉目标:LW10
MOVW   #A1张拉目标:LW10, #比较最小值:LW18
Network 11
LDW>=  #比较最小值:LW18, #A2张拉目标:LW14
MOVW   #A2张拉目标:LW14, #比较最小值:LW18
Network 12
LDW>=  #比较最小值:LW18, #B2张拉目标:LW16
MOVW   #B2张拉目标:LW16, #比较最小值:LW18
Network 13
LD     Always_On:SM0.0
MOVW   #比较最小值:LW18, #最小值:LW8
END_SUBROUTINE_BLOCK

SUBROUTINE_BLOCK 公共标志:SBR13
TITLE=子程序注释
VAR
临时伸长量:WORD;	// LW0 
END_VAR
BEGIN
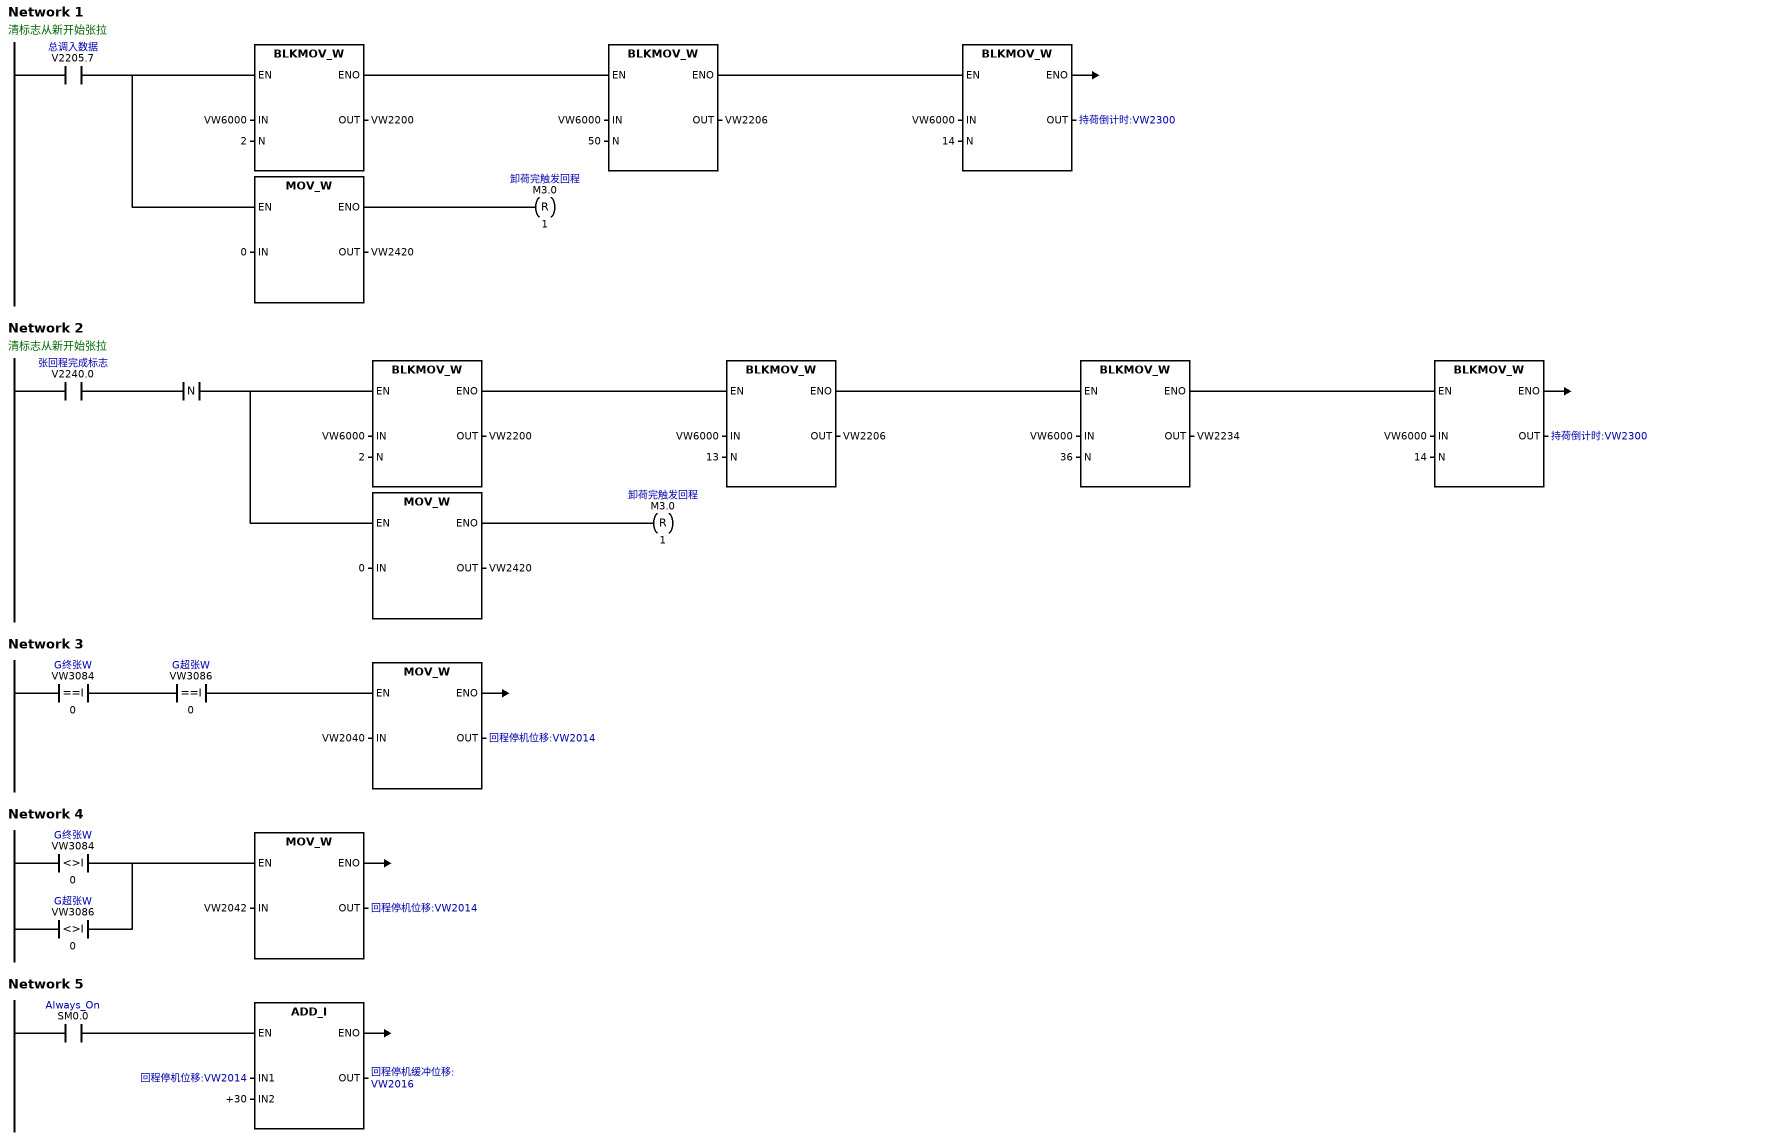
Network 1
// 清标志从新开始张拉
LD     总调入数据:V2205.7
LPS
BMW    VW6000, VW2200, 2
AENO
BMW    VW6000, VW2206, 50
AENO
BMW    VW6000, 持荷倒计时:VW2300, 14
LPP
MOVW   0, VW2420
AENO
R      卸荷完触发回程:M3.0, 1
Network 2
// 清标志从新开始张拉
LD     张回程完成标志:V2240.0
ED
LPS
BMW    VW6000, VW2200, 2
AENO
BMW    VW6000, VW2206, 13
AENO
BMW    VW6000, VW2234, 36
AENO
BMW    VW6000, 持荷倒计时:VW2300, 14
LPP
MOVW   0, VW2420
AENO
R      卸荷完触发回程:M3.0, 1
Network 3
LDW=   G终张W:VW3084, 0
AW=    G超张W:VW3086, 0
MOVW   VW2040, 回程停机位移:VW2014
Network 4
LDW<>  G终张W:VW3084, 0
OW<>   G超张W:VW3086, 0
MOVW   VW2042, 回程停机位移:VW2014
Network 5
LD     Always_On:SM0.0
MOVW   回程停机位移:VW2014, 回程停机缓冲位移:VW2016
+I     +30, 回程停机缓冲位移:VW2016
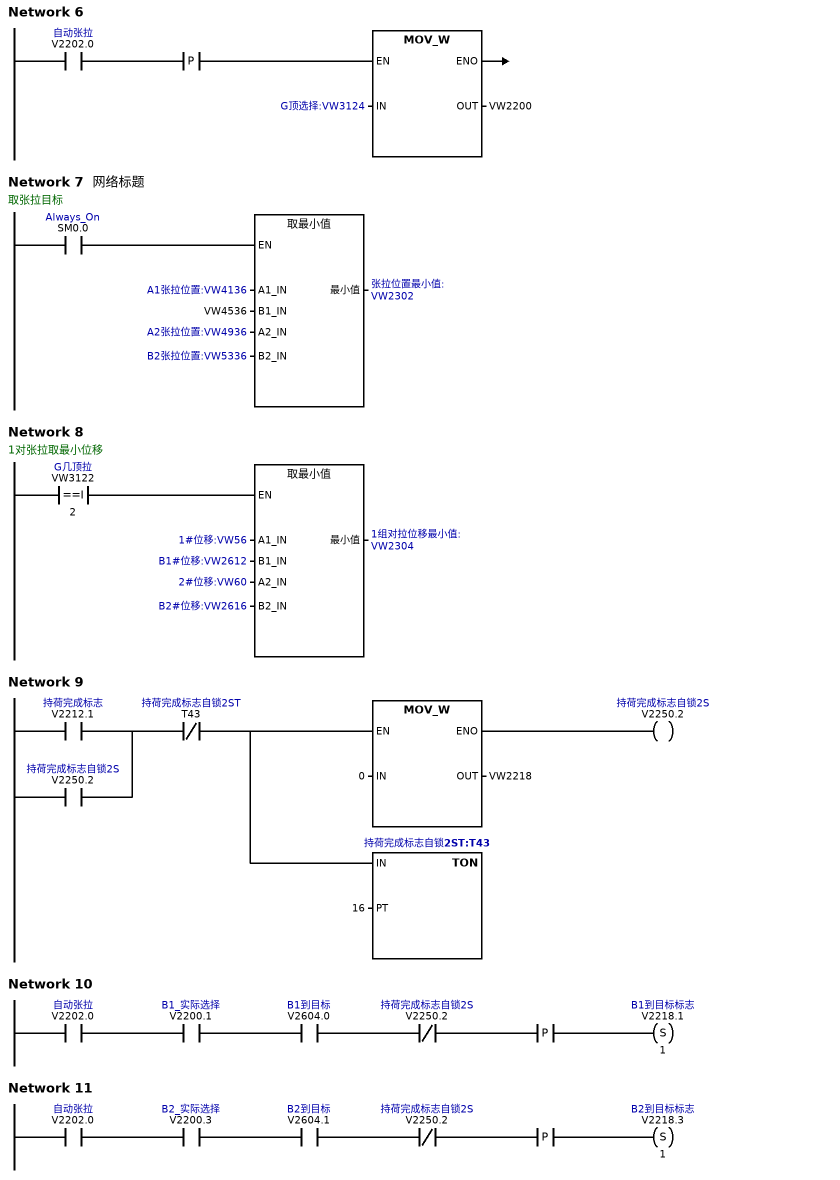
Network 6
LD     自动张拉:V2202.0
EU
MOVW   G顶选择:VW3124, VW2200
Network 7 // 网络标题
// 取张拉目标
LD     Always_On:SM0.0
CALL   取最小值:SBR12, A1张拉位置:VW4136, VW4536, A2张拉位置:VW4936, B2张拉位置:VW5336, 张拉位置最小值:VW2302
Network 8
// 1对张拉取最小位移
LDW=   G几顶拉:VW3122, 2
CALL   取最小值:SBR12, 1#位移:VW56, B1#位移:VW2612, 2#位移:VW60, B2#位移:VW2616, 1组对拉位移最小值:VW2304
Network 9
LD     持荷完成标志:V2212.1
O      持荷完成标志自锁2S:V2250.2
AN     持荷完成标志自锁2ST:T43
LPS
MOVW   0, VW2218
AENO
=      持荷完成标志自锁2S:V2250.2
LPP
TON    持荷完成标志自锁2ST:T43, 16
Network 10
LD     自动张拉:V2202.0
A      B1_实际选择:V2200.1
A      B1到目标:V2604.0
AN     持荷完成标志自锁2S:V2250.2
EU
S      B1到目标标志:V2218.1, 1
Network 11
LD     自动张拉:V2202.0
A      B2_实际选择:V2200.3
A      B2到目标:V2604.1
AN     持荷完成标志自锁2S:V2250.2
EU
S      B2到目标标志:V2218.3, 1
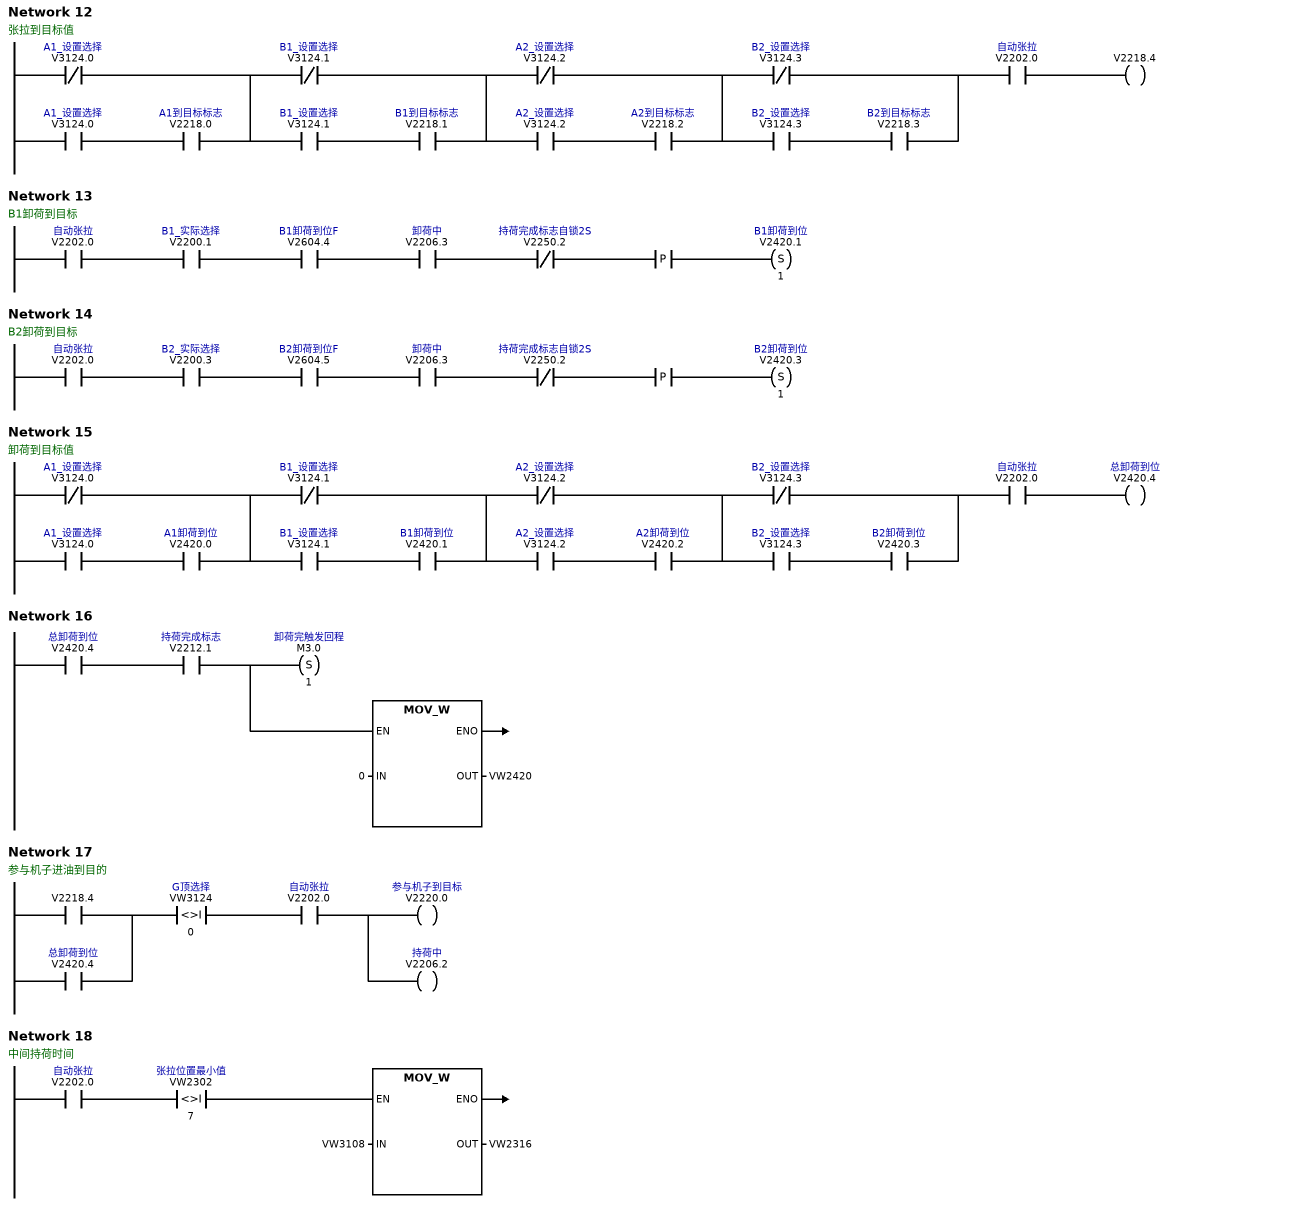
Network 12
// 张拉到目标值
LDN    A1_设置选择:V3124.0
LD     A1_设置选择:V3124.0
A      A1到目标标志:V2218.0
OLD
LDN    B1_设置选择:V3124.1
LD     B1_设置选择:V3124.1
A      B1到目标标志:V2218.1
OLD
ALD
LDN    A2_设置选择:V3124.2
LD     A2_设置选择:V3124.2
A      A2到目标标志:V2218.2
OLD
ALD
LDN    B2_设置选择:V3124.3
LD     B2_设置选择:V3124.3
A      B2到目标标志:V2218.3
OLD
ALD
A      自动张拉:V2202.0
=      V2218.4
Network 13
// B1卸荷到目标
LD     自动张拉:V2202.0
A      B1_实际选择:V2200.1
A      B1卸荷到位F:V2604.4
A      卸荷中:V2206.3
AN     持荷完成标志自锁2S:V2250.2
EU
S      B1卸荷到位:V2420.1, 1
Network 14
// B2卸荷到目标
LD     自动张拉:V2202.0
A      B2_实际选择:V2200.3
A      B2卸荷到位F:V2604.5
A      卸荷中:V2206.3
AN     持荷完成标志自锁2S:V2250.2
EU
S      B2卸荷到位:V2420.3, 1
Network 15
// 卸荷到目标值
LDN    A1_设置选择:V3124.0
LD     A1_设置选择:V3124.0
A      A1卸荷到位:V2420.0
OLD
LDN    B1_设置选择:V3124.1
LD     B1_设置选择:V3124.1
A      B1卸荷到位:V2420.1
OLD
ALD
LDN    A2_设置选择:V3124.2
LD     A2_设置选择:V3124.2
A      A2卸荷到位:V2420.2
OLD
ALD
LDN    B2_设置选择:V3124.3
LD     B2_设置选择:V3124.3
A      B2卸荷到位:V2420.3
OLD
ALD
A      自动张拉:V2202.0
=      总卸荷到位:V2420.4
Network 16
LD     总卸荷到位:V2420.4
A      持荷完成标志:V2212.1
S      卸荷完触发回程:M3.0, 1
MOVW   0, VW2420
Network 17
// 参与机子进油到目的
LD     V2218.4
O      总卸荷到位:V2420.4
AW<>   G顶选择:VW3124, 0
A      自动张拉:V2202.0
=      参与机子到目标:V2220.0
=      持荷中:V2206.2
Network 18
// 中间持荷时间
LD     自动张拉:V2202.0
AW<>   张拉位置最小值:VW2302, 7
MOVW   VW3108, VW2316
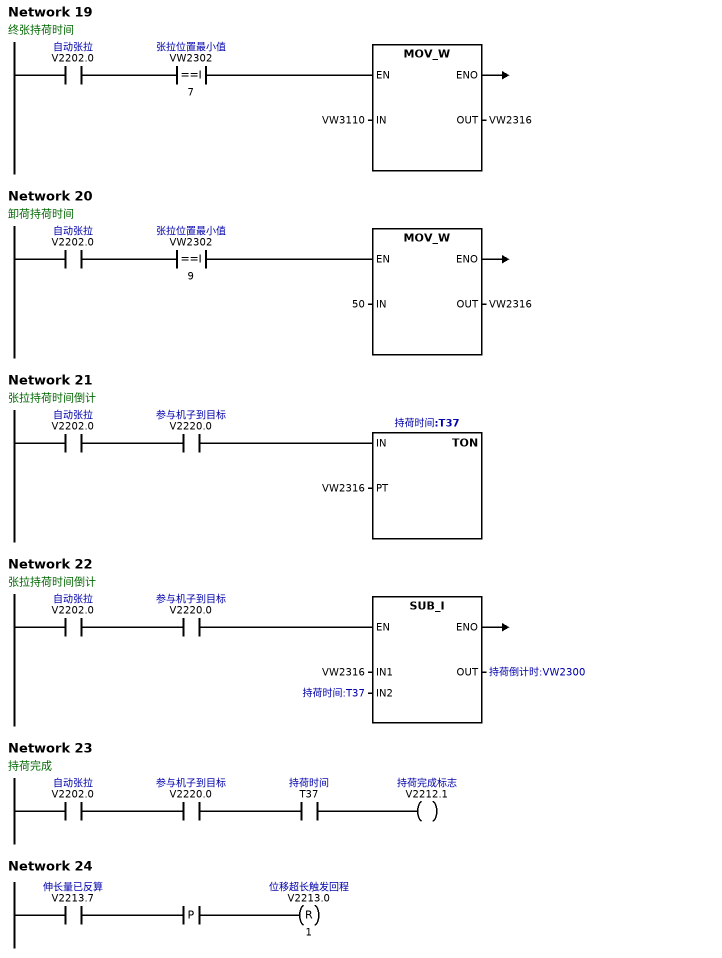
Network 19
// 终张持荷时间
LD     自动张拉:V2202.0
AW=    张拉位置最小值:VW2302, 7
MOVW   VW3110, VW2316
Network 20
// 卸荷持荷时间
LD     自动张拉:V2202.0
AW=    张拉位置最小值:VW2302, 9
MOVW   50, VW2316
Network 21
// 张拉持荷时间倒计
LD     自动张拉:V2202.0
A      参与机子到目标:V2220.0
TON    持荷时间:T37, VW2316
Network 22
// 张拉持荷时间倒计
LD     自动张拉:V2202.0
A      参与机子到目标:V2220.0
MOVW   VW2316, 持荷倒计时:VW2300
-I     持荷时间:T37, 持荷倒计时:VW2300
Network 23
// 持荷完成
LD     自动张拉:V2202.0
A      参与机子到目标:V2220.0
A      持荷时间:T37
=      持荷完成标志:V2212.1
Network 24
LD     伸长量已反算:V2213.7
EU
R      位移超长触发回程:V2213.0, 1
